(* IEC 61131-3 sources: std_i2980_v2.06_cp053/Source/IMM/ieccontrol/simulation (part 3) *)

(* ---- ABEasyMoldSimu.pu ---- *)
IMPORT_OVER_LISTFILE
 GET_REFTO
, EasyMold_Cmd
, tsCutOffCriterions

END_IMPORT

ALGORITHM_BLOCK ABEasyMoldSimu #DUMMY_EDIT_BLOCK

SYSTEM_VAR
 sv_MoldFullPosition : REAL;
 sv_MaxPressureSimu : REAL;
 sv_bAutoCycleRunning : BOOL;
 sv_ipCmd : REFTO EasyMold_Cmd;
 sv_CutOffParams : tsCutOffCriterions;
 sv_rScrewVolume : REAL;
 sv_rScrewDiameter : REAL;
 sv_rScrewPosition : REAL;
 sv_bEasyMoldTest : BOOL;
END_VAR

SYSTEM_OBJECT
 TaskSlow : TASK;
END_OBJECT

VAR
 uCounter : UDINT;
 rSAFactor : REAL;
 uTestCounter : UDINT := 0;
END_VAR

ALGORITHM EasyMoldWizardTest1

VAR_INPUT
 bRestart : BOOL := FALSE;
END_VAR

VAR_OUTPUT
 bReady : BOOL := FALSE;
END_VAR

VAR
 uCyclicCounter : UDINT := 0;
 uCyclicCounterPost : UDINT := 0;
 uCyclicLimit : UDINT := 2;
 uCyclicLimitTemp : UDINT := 2;
 rMaxPressSimu : REAL := 0.25;
 rMaxPressSimuPressLimit : REAL := 0.95;
 rDeltaPos : REAL := 0.0;
 rMoldFullPositionStart : REAL := 0.8;
 rMoldFullPositionStart1 : REAL := 0.2;
END_VAR
#BEGIN_EDIT_BLOCK
IF (rSAFactor <= 0.0) THEN
   rSAFactor := 1.0;
END_IF;
IF sv_rScrewVolume <= 0.0 THEN
   sv_MoldFullPosition :=  0.0;
   sv_MaxPressureSimu  :=  0.0;
   RETURN;
END_IF;
IF bRestart THEN
      bReady := FALSE;
      sv_MoldFullPosition := 0.001;//2.0 * sv_rScrewDiameter * 0.1 / sv_rScrewVolume;
      sv_MaxPressureSimu  := 0.05;
      uCyclicCounter      := 0;
      rDeltaPos           := 0.0;
ELSE
   IF sv_bAutoCycleRunning THEN

      CASE sv_ipCmd^ OF

         EMOLD_CMD_START: // Start
            bReady := FALSE;
            sv_MoldFullPosition := rMoldFullPositionStart;
            sv_MaxPressureSimu  :=  rMaxPressSimu;

         EMOLD_CMD_START1: // Start1
            sv_MoldFullPosition :=   rMoldFullPositionStart1;
            IF sv_MoldFullPosition >= ((sv_CutOffParams.rPositionThreshold / sv_rScrewVolume)- 0.1) THEN
                sv_MoldFullPosition := (sv_CutOffParams.rPositionThreshold - 0.11 * sv_rScrewVolume) / sv_rScrewVolume;
            END_IF;
            sv_MaxPressureSimu  :=  rMaxPressSimu;

         EMOLD_CMD_OPTIMIZE: // Optimize
            sv_MoldFullPosition :=  (sv_CutOffParams.rPositionThreshold - 0.01 * sv_rScrewVolume) / sv_rScrewVolume;
            IF sv_MoldFullPosition > rMoldFullPositionStart1 THEN
                rDeltaPos := sv_MoldFullPosition - rMoldFullPositionStart1;
                sv_MoldFullPosition := rMoldFullPositionStart1;
            END_IF;
            sv_MaxPressureSimu  :=  rMaxPressSimu;
            uCyclicCounter      :=  0;
            uCyclicCounterPost  := 0;

         EMOLD_CMD_CYCL_INJ:
//            IF uCyclicCounter = 0 THEN // 4
//               sv_MoldFullPosition := (0.95 * sv_rScrewVolume) / sv_rScrewVolume;
//               sv_MaxPressureSimu  := rMaxPressSimu;
//            ELSIF uCyclicCounter < uCyclicLimit THEN // 4
//               sv_MoldFullPosition := (sv_CutOffParams.rPositionThreshold + 0.01 * sv_rScrewVolume)  / sv_rScrewVolume;
//               sv_MaxPressureSimu  := rMaxPressSimu;
            IF uCyclicCounter = 0 THEN
               sv_MoldFullPosition := (sv_CutOffParams.rPositionThreshold - 0.01 * sv_rScrewVolume)  / sv_rScrewVolume - rDeltaPos;
               sv_MaxPressureSimu  := rMaxPressSimu;
            ELSIF uCyclicCounter < uCyclicLimit THEN
               sv_MoldFullPosition := (sv_CutOffParams.rPositionThreshold + 0.01 * sv_rScrewVolume)  / sv_rScrewVolume;
               sv_MaxPressureSimu  := rMaxPressSimuPressLimit;
            ELSIF uCyclicCounter < uCyclicLimit+uCyclicLimitTemp THEN
               sv_MoldFullPosition := (sv_CutOffParams.rPositionThreshold + 0.01 * sv_rScrewVolume)  / sv_rScrewVolume;
               sv_MaxPressureSimu  := rMaxPressSimu;
            ELSE
               sv_MoldFullPosition := (sv_CutOffParams.rPositionThreshold - 0.01 * sv_rScrewVolume)  / sv_rScrewVolume - rDeltaPos;
               sv_MaxPressureSimu  := rMaxPressSimu;
            END_IF;
            uCyclicCounter := uCyclicCounter +1;

         EMOLD_CMD_INC_MELTTEMP: //
            sv_MoldFullPosition := (sv_CutOffParams.rPositionThreshold - 0.01 * sv_rScrewVolume) / sv_rScrewVolume - rDeltaPos;
            sv_MaxPressureSimu  := rMaxPressSimu;

         EMOLD_CMD_INC_MOLDTEMP: // CyclicInject 1: 1. Durchlauf
            sv_MoldFullPosition := (sv_CutOffParams.rPositionThreshold - 0.01 * sv_rScrewVolume) / sv_rScrewVolume - rDeltaPos;
            sv_MaxPressureSimu  := rMaxPressSimu;

         EMOLD_CMD_POSTCUTOFF:
//            IF (uCyclicCounterPost=0) THEN
//               sv_MoldFullPosition := (0.95 * sv_rScrewVolume) / sv_rScrewVolume;
//               sv_MaxPressureSimu  := rMaxPressSimu;
//               uCyclicCounter      :=  0;
//                uCyclicCounterPost := 1;
//            ELSE
                sv_MoldFullPosition := (sv_CutOffParams.rPositionThreshold - 0.01 * sv_rScrewVolume) / sv_rScrewVolume - rDeltaPos;
                sv_MaxPressureSimu  := rMaxPressSimu;
                uCyclicCounter      := 0;
//            END_IF;

         EMOLD_CMD_INC_PACKPRESS:
            sv_MoldFullPosition := (sv_CutOffParams.rPositionThreshold - 0.01 * sv_rScrewVolume) / sv_rScrewVolume - rDeltaPos;
            sv_MaxPressureSimu  := rMaxPressSimuPressLimit;

         EMOLD_CMD_CORR_MELTCUS:
            sv_MoldFullPosition := (sv_CutOffParams.rPositionThreshold - 0.01 * sv_rScrewVolume) / sv_rScrewVolume - rDeltaPos;
            sv_MaxPressureSimu  := rMaxPressSimu;
            bReady := TRUE;

         EMOLD_CMD_HOTRUNNER: //
            sv_MoldFullPosition := (sv_CutOffParams.rPositionThreshold - 0.01 * sv_rScrewVolume) / sv_rScrewVolume - rDeltaPos;
            sv_MaxPressureSimu  := rMaxPressSimu;

      ELSE
            // default state
            bReady := FALSE;
            sv_MoldFullPosition := (sv_CutOffParams.rPositionThreshold - 0.01 * sv_rScrewVolume) / sv_rScrewVolume - rDeltaPos;
            sv_MaxPressureSimu  := rMaxPressSimu;

      END_CASE;
      uCounter := uCounter+1;
   ELSE
      sv_MoldFullPosition := sv_rScrewDiameter * 0.1 / sv_rScrewVolume;
      sv_MaxPressureSimu  := 50.0;
   END_IF;
   IF (sv_MoldFullPosition < 0.001) THEN
       sv_MoldFullPosition := 0.001;
   END_IF;
END_IF;
IF sv_MoldFullPosition > 1.0 THEN
   sv_MoldFullPosition := 1.0;
END_IF;

;#END_EDIT_BLOCK END_ALGORITHM

POSTUPDATE_ALGORITHM puEasyMoldWizardTestStart ON TaskSlow WITH sv_bEasyMoldTest

#BEGIN_EDIT_BLOCK

IF sv_bEasyMoldTest THEN
   uCounter := 1;
   rSAFactor := sv_rScrewDiameter * sv_rScrewDiameter * cEMW_Pi * 0.25e-3;
   sv_rScrewPosition := sv_rScrewDiameter * rSAFactor;
   uTestCounter := 0;
   START_PROCESS_ALGORITHM(paRunAlgo);
END_IF;

;#END_EDIT_BLOCK END_ALGORITHM

POSTUPDATE_ALGORITHM puEasyMoldWizardTestRun ON TaskSlow WITH sv_bAutoCycleRunning

#BEGIN_EDIT_BLOCK
IF sv_bEasyMoldTest THEN
    //piCmd := @sv_iCmd;
    START_PROCESS_ALGORITHM(paRunAlgo);
END_IF;

;#END_EDIT_BLOCK END_ALGORITHM

PROCESS_ALGORITHM paRunAlgo ON TaskSlow

#BEGIN_EDIT_BLOCK
CASE uTestCounter OF
   0:
      EasyMoldWizardTest1(bRestart:=TRUE);
      uTestCounter := uTestCounter + 1;

   1: // EasyMoldWizardTest1
      EasyMoldWizardTest1(bRestart:=FALSE);

ELSE
   // EasyMoldWizardTest1
   EasyMoldWizardTest1();
   uTestCounter := 1;
END_CASE;

STOP_PROCESS_ALGORITHM();

;#END_EDIT_BLOCK END_ALGORITHM

END_ALGORITHM_BLOCK

#END_OF_IEC_PART

@Puma @IecEditor 6 97 @Pou 25
@@@BEG_Comment@@@

@@@END_Comment@@@

@BEG_Contents

@BEG_Func
@RT(17)FuncTreeContainer
1
@Var @RT(9)GET_REFTO @RT(0) @T @T @DERIVED 0 @F @RT(22)KEBA_STANDARD_FUNCTION @F
@T
@BEG_Attrib
0 @RT(0) @RT(0)
@END_Attrib
1 1 @F @F @F @F

@END_Func

@BEG_Const
@RT(18)ConstTreeContainer
0
@END_Const

@BEG_Export

@BEG_Kind
@ALGORITHM_BLOCK @RT(14)ABEasyMoldSimu @STRUCTURED_TEXT
@RT(0) @RT(0) @RT(0)
@END_Kind

@BEG_Dcl
@RT(16)DclTreeContainer
13
@Var @RT(8)TaskSlow @RT(0) @T @F @DT @RT(4)TASK @RT(0) @T @T @BASIC 0 @F
@F @F
@T
@BEG_Attrib
3 @RT(0) @RT(0) @RT(0)
@END_Attrib
1 7 @F @F @F @F

@Var @RT(19)sv_MoldFullPosition @RT(0) @T @F @DT @RT(4)REAL @RT(0) @T @T @BASIC 0 @F
@F @F
@T
@BEG_Attrib
3 @RT(0) @RT(0) @RT(0)
@END_Attrib
1 8 @F @F @F @F

@Var @RT(18)sv_MaxPressureSimu @RT(0) @T @F @DT @RT(4)REAL @RT(0) @T @T @BASIC 0 @F
@F @F
@T
@BEG_Attrib
3 @RT(0) @RT(0) @RT(0)
@END_Attrib
1 8 @F @F @F @F

@Var @RT(20)sv_bAutoCycleRunning @RT(0) @T @F @DT @RT(4)BOOL @RT(0) @T @T @BASIC 0 @F
@F @F
@T
@BEG_Attrib
3 @RT(0) @RT(0) @RT(0)
@END_Attrib
1 8 @F @F @F @F

@Var @RT(8)sv_ipCmd @RT(0) @T @T @REFTO 0 @F @DERIVED 0 @T @T @DT @RT(12)EasyMold_Cmd @RT(0) @T @T @UNKNOWN 0 @F
@F @F
@T
@BEG_Attrib
3 @RT(0) @RT(0) @RT(0)
@END_Attrib
1 8 @F @F @F @F

@Var @RT(15)sv_CutOffParams @RT(0) @T @T @DERIVED 0 @T @T @DT @RT(18)tsCutOffCriterions @RT(0) @T @T @UNKNOWN 0 @F
@F @F
@T
@BEG_Attrib
3 @RT(0) @RT(0) @RT(0)
@END_Attrib
1 8 @F @F @F @F

@Var @RT(15)sv_rScrewVolume @RT(0) @T @F @DT @RT(4)REAL @RT(0) @T @T @BASIC 0 @F
@F @F
@T
@BEG_Attrib
3 @RT(0) @RT(0) @RT(0)
@END_Attrib
1 8 @F @F @F @F

@Var @RT(8)uCounter @RT(0) @T @F @DT @RT(5)UDINT @RT(0) @T @T @BASIC 0 @F
@F @F
@T
@BEG_Attrib
3 @RT(0) @RT(0) @RT(0)
@END_Attrib
1 0 @F @F @F @F

@Var @RT(17)sv_rScrewDiameter @RT(0) @T @F @DT @RT(4)REAL @RT(0) @T @T @BASIC 0 @F
@F @F
@T
@BEG_Attrib
3 @RT(0) @RT(0) @RT(0)
@END_Attrib
1 8 @F @F @F @F

@Var @RT(9)rSAFactor @RT(0) @T @F @DT @RT(4)REAL @RT(0) @T @T @BASIC 0 @F
@F @F
@T
@BEG_Attrib
3 @RT(0) @RT(0) @RT(0)
@END_Attrib
1 0 @F @F @F @F

@Var @RT(17)sv_rScrewPosition @RT(0) @T @F @DT @RT(4)REAL @RT(0) @T @T @BASIC 0 @F
@F @F
@T
@BEG_Attrib
3 @RT(0) @RT(0) @RT(0)
@END_Attrib
1 8 @F @F @F @F

@Var @RT(16)sv_bEasyMoldTest @RT(0) @T @F @DT @RT(4)BOOL @RT(0) @T @T @BASIC 0 @F
@F @F
@T
@BEG_Attrib
3 @RT(0) @RT(0) @RT(0)
@END_Attrib
1 8 @F @F @F @F

@Var @RT(12)uTestCounter @RT(0) @T @F @DT @RT(5)UDINT @RT(0) @T @T @BASIC 0 @F
@F @F
@T
@BEG_Attrib
3 @RT(1)0 @RT(0) @RT(0)
@END_Attrib
1 0 @F @F @F @F

@END_Dcl

@END_Export

@BEG_Body

4

@BEG_Export

@BEG_Algo
@ALGORITHM @RT(19)EasyMoldWizardTest1 @STRUCTURED_TEXT
@RT(0) @RT(0) @RT(0) @F @F
@END_Algo

@BEG_Dcl
@RT(16)DclTreeContainer
11
@Var @RT(8)bRestart @RT(0) @T @F @DT @RT(4)BOOL @RT(0) @T @T @BASIC 0 @F
@F @F
@T
@BEG_Attrib
3 @RT(5)FALSE @RT(0) @RT(0)
@END_Attrib
1 1 @F @F @F @F

@Var @RT(6)bReady @RT(0) @T @F @DT @RT(4)BOOL @RT(0) @T @T @BASIC 0 @F
@F @F
@T
@BEG_Attrib
3 @RT(5)FALSE @RT(0) @RT(0)
@END_Attrib
1 3 @F @F @F @F

@Var @RT(14)uCyclicCounter @RT(0) @T @F @DT @RT(5)UDINT @RT(0) @T @T @BASIC 0 @F
@F @F
@T
@BEG_Attrib
3 @RT(1)0 @RT(0) @RT(0)
@END_Attrib
1 0 @F @F @F @F

@Var @RT(18)uCyclicCounterPost @RT(0) @T @F @DT @RT(5)UDINT @RT(0) @T @T @BASIC 0 @F
@F @F
@T
@BEG_Attrib
3 @RT(1)0 @RT(0) @RT(0)
@END_Attrib
1 0 @F @F @F @F

@Var @RT(12)uCyclicLimit @RT(0) @T @F @DT @RT(5)UDINT @RT(0) @T @T @BASIC 0 @F
@F @F
@T
@BEG_Attrib
3 @RT(1)2 @RT(0) @RT(0)
@END_Attrib
1 0 @F @F @F @F

@Var @RT(16)uCyclicLimitTemp @RT(0) @T @F @DT @RT(5)UDINT @RT(0) @T @T @BASIC 0 @F
@F @F
@T
@BEG_Attrib
3 @RT(1)2 @RT(0) @RT(0)
@END_Attrib
1 0 @F @F @F @F

@Var @RT(13)rMaxPressSimu @RT(0) @T @F @DT @RT(4)REAL @RT(0) @T @T @BASIC 0 @F
@F @F
@T
@BEG_Attrib
3 @RT(4)0.25 @RT(0) @RT(0)
@END_Attrib
1 0 @F @F @F @F

@Var @RT(23)rMaxPressSimuPressLimit @RT(0) @T @F @DT @RT(4)REAL @RT(0) @T @T @BASIC 0 @F
@F @F
@T
@BEG_Attrib
3 @RT(4)0.95 @RT(0) @RT(0)
@END_Attrib
1 0 @F @F @F @F

@Var @RT(9)rDeltaPos @RT(0) @T @F @DT @RT(4)REAL @RT(0) @T @T @BASIC 0 @F
@F @F
@T
@BEG_Attrib
3 @RT(3)0.0 @RT(0) @RT(0)
@END_Attrib
1 0 @F @F @F @F

@Var @RT(22)rMoldFullPositionStart @RT(0) @T @F @DT @RT(4)REAL @RT(0) @T @T @BASIC 0 @F
@F @F
@T
@BEG_Attrib
3 @RT(3)0.8 @RT(0) @RT(0)
@END_Attrib
1 0 @F @F @F @F

@Var @RT(23)rMoldFullPositionStart1 @RT(0) @T @F @DT @RT(4)REAL @RT(0) @T @T @BASIC 0 @F
@F @F
@T
@BEG_Attrib
3 @RT(3)0.2 @RT(0) @RT(0)
@END_Attrib
1 0 @F @F @F @F

@END_Dcl

@END_Export

@BEG_Export

@BEG_Algo
@POSTUPDATE_ALGORITHM @RT(25)puEasyMoldWizardTestStart @STRUCTURED_TEXT
@RT(0) @RT(16)sv_bEasyMoldTest @RT(8)TaskSlow @F @F
@END_Algo

@BEG_Dcl
@RT(16)DclTreeContainer
0
@END_Dcl

@END_Export

@BEG_Export

@BEG_Algo
@POSTUPDATE_ALGORITHM @RT(23)puEasyMoldWizardTestRun @STRUCTURED_TEXT
@RT(0) @RT(20)sv_bAutoCycleRunning @RT(8)TaskSlow @F @F
@END_Algo

@BEG_Dcl
@RT(16)DclTreeContainer
0
@END_Dcl

@END_Export

@BEG_Export

@BEG_Algo
@PROCESS_ALGORITHM @RT(9)paRunAlgo @STRUCTURED_TEXT
@RT(0) @RT(0) @RT(8)TaskSlow @F @F
@END_Algo

@BEG_Dcl
@RT(16)DclTreeContainer
0
@END_Dcl

@END_Export

@BEG_Body
@TL(117)
IF (rSAFactor <= 0.0) THEN
   rSAFactor := 1.0;
END_IF;
IF sv_rScrewVolume <= 0.0 THEN
   sv_MoldFullPosition :=  0.0;
   sv_MaxPressureSimu  :=  0.0;
   RETURN;
END_IF;
IF bRestart THEN
      bReady := FALSE;
      sv_MoldFullPosition := 0.001;//2.0 * sv_rScrewDiameter * 0.1 / sv_rScrewVolume;
      sv_MaxPressureSimu  := 0.05;
      uCyclicCounter      := 0;
      rDeltaPos           := 0.0;
ELSE
   IF sv_bAutoCycleRunning THEN

      CASE sv_ipCmd^ OF

         EMOLD_CMD_START: // Start
            bReady := FALSE;
            sv_MoldFullPosition := rMoldFullPositionStart;
            sv_MaxPressureSimu  :=  rMaxPressSimu;

         EMOLD_CMD_START1: // Start1
            sv_MoldFullPosition :=   rMoldFullPositionStart1;
            IF sv_MoldFullPosition >= ((sv_CutOffParams.rPositionThreshold / sv_rScrewVolume)- 0.1) THEN
                sv_MoldFullPosition := (sv_CutOffParams.rPositionThreshold - 0.11 * sv_rScrewVolume) / sv_rScrewVolume;
            END_IF;
            sv_MaxPressureSimu  :=  rMaxPressSimu;

         EMOLD_CMD_OPTIMIZE: // Optimize
            sv_MoldFullPosition :=  (sv_CutOffParams.rPositionThreshold - 0.01 * sv_rScrewVolume) / sv_rScrewVolume;
            IF sv_MoldFullPosition > rMoldFullPositionStart1 THEN
                rDeltaPos := sv_MoldFullPosition - rMoldFullPositionStart1;
                sv_MoldFullPosition := rMoldFullPositionStart1;
            END_IF;
            sv_MaxPressureSimu  :=  rMaxPressSimu;
            uCyclicCounter      :=  0;
            uCyclicCounterPost  := 0;

         EMOLD_CMD_CYCL_INJ:
//            IF uCyclicCounter = 0 THEN // 4
//               sv_MoldFullPosition := (0.95 * sv_rScrewVolume) / sv_rScrewVolume;
//               sv_MaxPressureSimu  := rMaxPressSimu;
//            ELSIF uCyclicCounter < uCyclicLimit THEN // 4
//               sv_MoldFullPosition := (sv_CutOffParams.rPositionThreshold + 0.01 * sv_rScrewVolume)  / sv_rScrewVolume;
//               sv_MaxPressureSimu  := rMaxPressSimu;
            IF uCyclicCounter = 0 THEN
               sv_MoldFullPosition := (sv_CutOffParams.rPositionThreshold - 0.01 * sv_rScrewVolume)  / sv_rScrewVolume - rDeltaPos;
               sv_MaxPressureSimu  := rMaxPressSimu;
            ELSIF uCyclicCounter < uCyclicLimit THEN
               sv_MoldFullPosition := (sv_CutOffParams.rPositionThreshold + 0.01 * sv_rScrewVolume)  / sv_rScrewVolume;
               sv_MaxPressureSimu  := rMaxPressSimuPressLimit;
            ELSIF uCyclicCounter < uCyclicLimit+uCyclicLimitTemp THEN
               sv_MoldFullPosition := (sv_CutOffParams.rPositionThreshold + 0.01 * sv_rScrewVolume)  / sv_rScrewVolume;
               sv_MaxPressureSimu  := rMaxPressSimu;
            ELSE
               sv_MoldFullPosition := (sv_CutOffParams.rPositionThreshold - 0.01 * sv_rScrewVolume)  / sv_rScrewVolume - rDeltaPos;
               sv_MaxPressureSimu  := rMaxPressSimu;
            END_IF;
            uCyclicCounter := uCyclicCounter +1;

         EMOLD_CMD_INC_MELTTEMP: //
            sv_MoldFullPosition := (sv_CutOffParams.rPositionThreshold - 0.01 * sv_rScrewVolume) / sv_rScrewVolume - rDeltaPos;
            sv_MaxPressureSimu  := rMaxPressSimu;

         EMOLD_CMD_INC_MOLDTEMP: // CyclicInject 1: 1. Durchlauf
            sv_MoldFullPosition := (sv_CutOffParams.rPositionThreshold - 0.01 * sv_rScrewVolume) / sv_rScrewVolume - rDeltaPos;
            sv_MaxPressureSimu  := rMaxPressSimu;

         EMOLD_CMD_POSTCUTOFF:
//            IF (uCyclicCounterPost=0) THEN
//               sv_MoldFullPosition := (0.95 * sv_rScrewVolume) / sv_rScrewVolume;
//               sv_MaxPressureSimu  := rMaxPressSimu;
//               uCyclicCounter      :=  0;
//                uCyclicCounterPost := 1;
//            ELSE
                sv_MoldFullPosition := (sv_CutOffParams.rPositionThreshold - 0.01 * sv_rScrewVolume) / sv_rScrewVolume - rDeltaPos;
                sv_MaxPressureSimu  := rMaxPressSimu;
                uCyclicCounter      := 0;
//            END_IF;

         EMOLD_CMD_INC_PACKPRESS:
            sv_MoldFullPosition := (sv_CutOffParams.rPositionThreshold - 0.01 * sv_rScrewVolume) / sv_rScrewVolume - rDeltaPos;
            sv_MaxPressureSimu  := rMaxPressSimuPressLimit;

         EMOLD_CMD_CORR_MELTCUS:
            sv_MoldFullPosition := (sv_CutOffParams.rPositionThreshold - 0.01 * sv_rScrewVolume) / sv_rScrewVolume - rDeltaPos;
            sv_MaxPressureSimu  := rMaxPressSimu;
            bReady := TRUE;

         EMOLD_CMD_HOTRUNNER: //
            sv_MoldFullPosition := (sv_CutOffParams.rPositionThreshold - 0.01 * sv_rScrewVolume) / sv_rScrewVolume - rDeltaPos;
            sv_MaxPressureSimu  := rMaxPressSimu;

      ELSE
            // default state
            bReady := FALSE;
            sv_MoldFullPosition := (sv_CutOffParams.rPositionThreshold - 0.01 * sv_rScrewVolume) / sv_rScrewVolume - rDeltaPos;
            sv_MaxPressureSimu  := rMaxPressSimu;

      END_CASE;
      uCounter := uCounter+1;
   ELSE
      sv_MoldFullPosition := sv_rScrewDiameter * 0.1 / sv_rScrewVolume;
      sv_MaxPressureSimu  := 50.0;
   END_IF;
   IF (sv_MoldFullPosition < 0.001) THEN
       sv_MoldFullPosition := 0.001;
   END_IF;
END_IF;
IF sv_MoldFullPosition > 1.0 THEN
   sv_MoldFullPosition := 1.0;
END_IF;

@END_Body

@@@BEG_Comment@@@
@TL(0)

@@@END_Comment@@@

@BEG_Body
@TL(9)

IF sv_bEasyMoldTest THEN
   uCounter := 1;
   rSAFactor := sv_rScrewDiameter * sv_rScrewDiameter * cEMW_Pi * 0.25e-3;
   sv_rScrewPosition := sv_rScrewDiameter * rSAFactor;
   uTestCounter := 0;
   START_PROCESS_ALGORITHM(paRunAlgo);
END_IF;

@END_Body

@@@BEG_Comment@@@
@TL(0)

@@@END_Comment@@@

@BEG_Body
@TL(5)
IF sv_bEasyMoldTest THEN
    //piCmd := @sv_iCmd;
    START_PROCESS_ALGORITHM(paRunAlgo);
END_IF;

@END_Body

@@@BEG_Comment@@@
@TL(0)

@@@END_Comment@@@

@BEG_Body
@TL(16)
CASE uTestCounter OF
   0:
      EasyMoldWizardTest1(bRestart:=TRUE);
      uTestCounter := uTestCounter + 1;

   1: // EasyMoldWizardTest1
      EasyMoldWizardTest1(bRestart:=FALSE);

ELSE
   // EasyMoldWizardTest1
   EasyMoldWizardTest1();
   uTestCounter := 1;
END_CASE;

STOP_PROCESS_ALGORITHM();

@END_Body

@@@BEG_Comment@@@
@TL(0)

@@@END_Comment@@@
@END_Body

@END_Contents

(* ---- ABEjeSimu.pu ---- *)
IMPORT_OVER_LISTFILE
 GET_TASK_INTERVAL
, GET_SYNC_REFTO
, KSYS_Status_OK
, FBEPForceAI
, FBEPForceDI
, FBEPUnForceAI
, FBEPUnForceDI
, tsRequiredPumps
, FBGetSimulationSource
, TON
, KSYS_Status
, FBGetRequiredPumps

END_IMPORT

ALGORITHM_BLOCK ABEjeSimu #DUMMY_EDIT_BLOCK

SYSTEM_VAR
 sv_bSimulate : BOOL;
 sv_bInitStart : BOOL;
 ai_Position_stat : BOOL;
 sv_ForceEjectorBack : BOOL;
 sv_bInitDone : BOOL;
END_VAR

SYSTEM_OBJECT
 TaskSim : TASK;
 PU_Task_13 : TASK;
 TaskAnalog : TASK;
END_OBJECT

VAR
 fbEPForceAI : FBEPForceAI;
 fbEPForceDI : FBEPForceDI;
 mbDIEjectorBackLinked : BOOL;
 fbEPUnForceAI : FBEPUnForceAI;
 fbEPUnForceDI : FBEPUnForceDI;
 mpPumps : REFTO tsRequiredPumps;
 mprVelocity : REFTO REAL;
 fbGetSimulationSource : FBGetSimulationSource;
END_VAR

POSTUPDATE_ALGORITHM pStart ON PU_Task_13 WITH sv_bSimulate,sv_bInitStart

#BEGIN_EDIT_BLOCK
(**************************************** WARNING ********************************************
 *** The KEBA Kemro K2 System including software is not intended for safety control tasks! ***
 ***                       For further information see Comment tab!                        ***
 *********************************************************************************************)

IF sv_bSimulate THEN
   START_PROCESS_ALGORITHM(paSimulate);
END_IF;

;#END_EDIT_BLOCK END_ALGORITHM

PROCESS_ALGORITHM paSimulate ON TaskAnalog

VAR
 rEjectDivision : REAL := 0.3;
 mrEjectorPosRaw : REAL;
 rEjectTimeFor10V : REAL := 1.0;
 TimerFwd : TON (* chad(CR_0038565) *);
 TimerBwd : TON (* chad(CR_0038565) *);
 rCycleTime : REAL;
 dCycleTime : TIME;
 prEjectorPosRaw : REFTO REAL;
 bAIEjectorTransLinked : BOOL;
 pbDOEjectorBwd : REFTO BOOL;
 pbDOEjectorFwd : REFTO BOOL;
 bDOEjectorFwdLinked : BOOL;
 bDOEjectorBwdLinked : BOOL;
 bDIEjectorFwdLinked : BOOL (* chad(CR_0038565) *);
 pbDummy : REFTO BOOL;
 Status : KSYS_Status;
 bDIEjectorSafetyPlateLinked : BOOL;
END_VAR

(* IecGraph-Code *)

(* init step *)
INITIAL_STEP INIT:
aInit (P);
END_STEP

(* steps *)
STEP SIM:
aSimulate (N);
END_STEP

STEP STOP:
aStopSimu (P);
END_STEP

(* transitions *)
TRANSITION SimRequired (* SimRequired *) FROM INIT TO SIM :=  #BEGIN_EDIT_BLOCK
sv_bSimulate
;#END_EDIT_BLOCK
END_TRANSITION

TRANSITION StpSimRequired (* StpSimRequired *) FROM SIM TO STOP :=  #BEGIN_EDIT_BLOCK
NOT sv_bSimulate
;#END_EDIT_BLOCK
END_TRANSITION

TRANSITION Return (* Return *) FROM STOP TO SIM :=  #BEGIN_EDIT_BLOCK
TRUE
;#END_EDIT_BLOCK
END_TRANSITION

(* end IecGraph-Code *)
(* sfc-code *)

(* stand alone actions *)
ACTION aInit: #BEGIN_EDIT_BLOCK
(**************************************** WARNING ********************************************
 *** The KEBA Kemro K2 System including software is not intended for safety control tasks! ***
 ***                       For further information see Comment tab!                        ***
 *********************************************************************************************)

pbDummy := GET_SYNC_REFTO('Ejector1.di_EjectorBwd', T#0s, Status);
mbDIEjectorBackLinked := (Status = KSYS_Status_OK);

pbDummy := GET_SYNC_REFTO('Ejector1.di_EjectorFwd', T#0s, Status);
bDIEjectorFwdLinked := (Status = KSYS_Status_OK);

prEjectorPosRaw := GET_SYNC_REFTO('Ejector1.ai_Position', T#0s, Status);
bAIEjectorTransLinked := (Status = KSYS_Status_OK);

pbDOEjectorFwd := GET_SYNC_REFTO('Ejector1.do_Forward', T#0s, Status);
bDOEjectorFwdLinked := (Status = KSYS_Status_OK);

pbDOEjectorBwd := GET_SYNC_REFTO('Ejector1.do_Backward', T#0s, Status);
bDOEjectorBwdLinked := (Status = KSYS_Status_OK);

pbDummy := GET_SYNC_REFTO('Ejector1.di_SafetyPlate', T#0s, Status);
bDIEjectorSafetyPlateLinked := (Status = KSYS_Status_OK);
IF bDIEjectorSafetyPlateLinked THEN
   fbEPForceDI(sSysVar := 'Ejector1.di_SafetyPlate',Value := TRUE);
END_IF;

dCycleTime :=  GET_TASK_INTERVAL();
rCycleTime := (LINT_TO_REAL(TIME_TO_LINT(dCycleTime))) / 1000000.0;
rEjectDivision := 1.0  / rEjectTimeFor10V * rCycleTime;

sv_ForceEjectorBack := TRUE;

IF bDIEjectorFwdLinked THEN    //chad(CR_0038565)
   fbEPForceDI(sSysVar := 'Ejector1.di_EjectorFwd',Value := FALSE);
END_IF;

IF bAIEjectorTransLinked THEN
   ai_Position_stat := FALSE;
   fbEPForceAI(sSysVar := 'Ejector1.ai_Position',Value := 0.0, Range := 10.0);
END_IF;

;#END_EDIT_BLOCK END_ACTION (*aInit*)
ACTION aSimulate: #BEGIN_EDIT_BLOCK
(**************************************** WARNING ********************************************
 *** The KEBA Kemro K2 System including software is not intended for safety control tasks! ***
 ***                       For further information see Comment tab!                        ***
 *********************************************************************************************)

IF bAIEjectorTransLinked THEN
   IF bDOEjectorFwdLinked AND pbDOEjectorFwd^ THEN
      mrEjectorPosRaw := prEjectorPosRaw^ + MUL(rEjectDivision,mprVelocity^);
      sv_ForceEjectorBack := FALSE;
   ELSIF bDOEjectorBwdLinked AND pbDOEjectorBwd^ THEN
      mrEjectorPosRaw := prEjectorPosRaw^ - MUL(rEjectDivision,mprVelocity^);
      IF prEjectorPosRaw^ <= 2.0 THEN
            sv_ForceEjectorBack := TRUE;
      END_IF;
   END_IF;
   fbEPForceAI(sSysVar := 'Ejector1.ai_Position', Value := MAX(mrEjectorPosRaw,0.0), Range := 10.0);

ELSE    //chad(CR_0038565) - transducer not linked

   //Move forward simulation
   IF bDOEjectorFwdLinked AND (NOT pbDOEjectorFwd^) THEN
      TimerFwd(IN := FALSE);
   END_IF;

   IF bDOEjectorFwdLinked AND pbDOEjectorFwd^ THEN
      TimerFwd(IN := TRUE, PT := t#4s);
      IF mbDIEjectorBackLinked THEN
         sv_ForceEjectorBack := FALSE;
         TimerBwd(IN := FALSE);
      END_IF;

      IF TimerFwd.Q AND bDIEjectorFwdLinked THEN
         fbEPForceDI(sSysVar := 'Ejector1.di_EjectorFwd',Value := TRUE);
         TimerFwd(IN := FALSE);
      END_IF;
   END_IF;

   //Move backward simulation
   IF bDOEjectorBwdLinked AND (NOT pbDOEjectorBwd^) THEN
      TimerBwd(IN := FALSE);
   END_IF;

   IF bDOEjectorBwdLinked AND pbDOEjectorBwd^ THEN
      TimerBwd(IN := TRUE, PT := t#4s);
      IF bDIEjectorFwdLinked THEN
         fbEPForceDI(sSysVar := 'Ejector1.di_EjectorFwd',Value := FALSE);
         TimerFwd(IN := FALSE);
      END_IF;

      IF TimerBwd.Q AND mbDIEjectorBackLinked THEN
         sv_ForceEjectorBack := TRUE;
         TimerBwd(IN := FALSE);
      END_IF;
   END_IF;
END_IF;

;#END_EDIT_BLOCK END_ACTION (*aSimulate*)
ACTION aStopSimu: #BEGIN_EDIT_BLOCK
(**************************************** WARNING ********************************************
 *** The KEBA Kemro K2 System including software is not intended for safety control tasks! ***
 ***                       For further information see Comment tab!                        ***
 *********************************************************************************************)

IF bAIEjectorTransLinked THEN
   fbEPUnForceAI(sSysVar := 'Ejector1.ai_Position');
END_IF;
IF mbDIEjectorBackLinked THEN
   fbEPUnForceDI(sSysVar := 'Ejector1.di_EjectorBwd');
END_IF;
IF bDIEjectorSafetyPlateLinked THEN
   fbEPUnForceDI(sSysVar := 'Ejector1.di_SafetyPlate');
END_IF;
IF bDIEjectorFwdLinked THEN   //chad(CR_0038565)
   fbEPUnForceDI(sSysVar := 'Ejector1.di_EjectorFwd');
END_IF;

STOP_PROCESS_ALGORITHM();

;#END_EDIT_BLOCK END_ACTION (*aStopSimu*)
(* end sfc-code *)

END_ALGORITHM

POSTUPDATE_ALGORITHM pEjectorBwd ON TaskSim WITH sv_ForceEjectorBack

#BEGIN_EDIT_BLOCK
(**************************************** WARNING ********************************************
 *** The KEBA Kemro K2 System including software is not intended for safety control tasks! ***
 ***                       For further information see Comment tab!                        ***
 *********************************************************************************************)

IF mbDIEjectorBackLinked THEN
   fbEPForceDI(sSysVar := 'Ejector1.di_EjectorBwd',Value := sv_ForceEjectorBack);
END_IF;

;#END_EDIT_BLOCK END_ALGORITHM

ALGORITHM aGetSimulationSource

#BEGIN_EDIT_BLOCK
(**************************************** WARNING ********************************************
 *** The KEBA Kemro K2 System including software is not intended for safety control tasks! ***
 ***                       For further information see Comment tab!                        ***
 *********************************************************************************************)

fbGetSimulationSource(pRequiredPumps := mpPumps,
                      prVelocity => mprVelocity);

;#END_EDIT_BLOCK END_ALGORITHM

POSTUPDATE_ALGORITHM pInitDone ON TaskSim WITH sv_bInitDone

VAR
 fbGetRequiredPumps : FBGetRequiredPumps;
END_VAR
#BEGIN_EDIT_BLOCK
(**************************************** WARNING ********************************************
 *** The KEBA Kemro K2 System including software is not intended for safety control tasks! ***
 ***                       For further information see Comment tab!                        ***
 *********************************************************************************************)

//get required pumps
fbGetRequiredPumps.DeviceId.CompId := cCompEjector;
fbGetRequiredPumps.DeviceId.IndexId := 1;

fbGetRequiredPumps(MoveDir := cMoveFwd,
                   MoveId := cMoveFwd);
mpPumps := fbGetRequiredPumps.pPumps;

aGetSimulationSource();

;#END_EDIT_BLOCK END_ALGORITHM

POSTUPDATE_ALGORITHM pRequiredPumps ON TaskSim WITH mpPumps^.RequiredPumps

#BEGIN_EDIT_BLOCK
(**************************************** WARNING ********************************************
 *** The KEBA Kemro K2 System including software is not intended for safety control tasks! ***
 ***                       For further information see Comment tab!                        ***
 *********************************************************************************************)

aGetSimulationSource();

;#END_EDIT_BLOCK END_ALGORITHM

END_ALGORITHM_BLOCK

#END_OF_IEC_PART

@Puma @IecEditor 6 113 @Pou 25
@@@BEG_Comment@@@

@@@END_Comment@@@

@BEG_Contents

@BEG_Func
@RT(17)FuncTreeContainer
2
@Var @RT(17)GET_TASK_INTERVAL @RT(0) @T @T @DERIVED 0 @F @RT(22)KEBA_STANDARD_FUNCTION @F
@T
@BEG_Attrib
0 @RT(0) @RT(0)
@END_Attrib
1 1 @F @F @F @F

@Var @RT(14)GET_SYNC_REFTO @RT(0) @T @T @DERIVED 0 @F @RT(22)KEBA_STANDARD_FUNCTION @F
@T
@BEG_Attrib
0 @RT(0) @RT(0)
@END_Attrib
1 1 @F @F @F @F

@END_Func

@BEG_Const
@RT(18)ConstTreeContainer
1
@Var @RT(14)KSYS_Status_OK @RT(0) @T @T @DERIVED 0 @F @RT(11)KSYS_Status @F
@T
@BEG_Attrib
0 @RT(1)1 @RT(0)
@END_Attrib
1 1 @F @F @F @F

@END_Const

@BEG_Export

@BEG_Kind
@ALGORITHM_BLOCK @RT(9)ABEjeSimu @STRUCTURED_TEXT
@RT(0) @RT(0) @RT(0)
@END_Kind

@BEG_Dcl
@RT(16)DclTreeContainer
16
@Var @RT(12)sv_bSimulate @RT(0) @T @F @DT @RT(4)BOOL @RT(0) @T @T @BASIC 0 @F
@F @F
@T
@BEG_Attrib
3 @RT(0) @RT(0) @RT(0)
@END_Attrib
1 8 @F @F @F @F

@Var @RT(13)sv_bInitStart @RT(0) @T @F @DT @RT(4)BOOL @RT(0) @T @T @BASIC 0 @F
@F @F
@T
@BEG_Attrib
3 @RT(0) @RT(0) @RT(0)
@END_Attrib
1 8 @F @F @F @F

@Var @RT(16)ai_Position_stat @RT(0) @T @F @DT @RT(4)BOOL @RT(0) @T @T @BASIC 0 @F
@F @F
@T
@BEG_Attrib
3 @RT(0) @RT(0) @RT(0)
@END_Attrib
1 8 @F @F @F @F

@Var @RT(7)TaskSim @RT(0) @T @F @DT @RT(4)TASK @RT(0) @T @T @BASIC 0 @F
@F @F
@T
@BEG_Attrib
3 @RT(0) @RT(0) @RT(0)
@END_Attrib
1 7 @F @F @F @F

@Var @RT(10)PU_Task_13 @RT(0) @T @F @DT @RT(4)TASK @RT(0) @T @T @BASIC 0 @F
@F @F
@T
@BEG_Attrib
3 @RT(0) @RT(0) @RT(0)
@END_Attrib
1 7 @F @F @F @F

@Var @RT(11)fbEPForceAI @RT(0) @T @T @DERIVED 0 @T @T @DT @RT(11)FBEPForceAI @RT(0) @T @T @UNKNOWN 0 @F
@F @F
@T
@BEG_Attrib
3 @RT(0) @RT(0) @RT(0)
@END_Attrib
1 0 @F @F @F @F

@Var @RT(11)fbEPForceDI @RT(0) @T @T @DERIVED 0 @T @T @DT @RT(11)FBEPForceDI @RT(0) @T @T @UNKNOWN 0 @F
@F @F
@T
@BEG_Attrib
3 @RT(0) @RT(0) @RT(0)
@END_Attrib
1 0 @F @F @F @F

@Var @RT(21)mbDIEjectorBackLinked @RT(0) @T @F @DT @RT(4)BOOL @RT(0) @T @T @BASIC 0 @F
@F @F
@T
@BEG_Attrib
3 @RT(0) @RT(0) @RT(0)
@END_Attrib
1 0 @F @F @F @F

@Var @RT(13)fbEPUnForceAI @RT(0) @T @T @DERIVED 0 @T @T @DT @RT(13)FBEPUnForceAI @RT(0) @T @T @UNKNOWN 0 @F
@F @F
@T
@BEG_Attrib
3 @RT(0) @RT(0) @RT(0)
@END_Attrib
1 0 @F @F @F @F

@Var @RT(13)fbEPUnForceDI @RT(0) @T @T @DERIVED 0 @T @T @DT @RT(13)FBEPUnForceDI @RT(0) @T @T @UNKNOWN 0 @F
@F @F
@T
@BEG_Attrib
3 @RT(0) @RT(0) @RT(0)
@END_Attrib
1 0 @F @F @F @F

@Var @RT(10)TaskAnalog @RT(0) @T @T @RENAMED 0 @T @T @DT @RT(4)TASK @RT(0) @T @T @BASIC 0 @F
@F @F
@T
@BEG_Attrib
3 @RT(0) @RT(0) @RT(0)
@END_Attrib
1 7 @F @F @F @F

@Var @RT(19)sv_ForceEjectorBack @RT(0) @T @T @RENAMED 0 @T @T @DT @RT(4)BOOL @RT(0) @T @T @BASIC 0 @F
@F @F
@T
@BEG_Attrib
3 @RT(0) @RT(0) @RT(0)
@END_Attrib
1 8 @F @F @F @F

@Var @RT(7)mpPumps @RT(0) @T @T @REFTO 0 @F @DERIVED 0 @T @T @DT @RT(15)tsRequiredPumps @RT(0) @T @T @UNKNOWN 0 @F
@F @F
@T
@BEG_Attrib
3 @RT(0) @RT(0) @RT(0)
@END_Attrib
1 0 @F @F @F @F

@Var @RT(12)sv_bInitDone @RT(0) @T @T @RENAMED 0 @T @T @DT @RT(4)BOOL @RT(0) @T @T @BASIC 0 @F
@F @F
@T
@BEG_Attrib
3 @RT(0) @RT(0) @RT(0)
@END_Attrib
1 8 @F @F @F @F

@Var @RT(11)mprVelocity @RT(0) @T @T @REFTO 0 @T @DT @RT(4)REAL @RT(0) @T @T @BASIC 0 @F
@F @F
@T
@BEG_Attrib
3 @RT(0) @RT(0) @RT(0)
@END_Attrib
1 0 @F @F @F @F

@Var @RT(21)fbGetSimulationSource @RT(0) @T @T @DERIVED 0 @T @T @DT @RT(21)FBGetSimulationSource @RT(0) @T @T @UNKNOWN 0 @F
@F @F
@T
@BEG_Attrib
3 @RT(0) @RT(0) @RT(0)
@END_Attrib
1 0 @F @F @F @F

@END_Dcl

@END_Export

@BEG_Body

6

@BEG_Export

@BEG_Algo
@POSTUPDATE_ALGORITHM @RT(6)pStart @STRUCTURED_TEXT
@RT(0) @RT(26)sv_bSimulate,sv_bInitStart @RT(10)PU_Task_13 @F @F
@END_Algo

@BEG_Dcl
@RT(16)DclTreeContainer
0
@END_Dcl

@END_Export

@BEG_Export

@BEG_Algo
@PROCESS_ALGORITHM @RT(10)paSimulate @SEQUENTIAL_FLOW_CHART
@RT(0) @RT(0) @RT(10)TaskAnalog @F @F
@END_Algo

@BEG_Dcl
@RT(16)DclTreeContainer
17
@Var @RT(14)rEjectDivision @RT(0) @T @F @DT @RT(4)REAL @RT(0) @T @T @BASIC 0 @F
@F @F
@T
@BEG_Attrib
3 @RT(3)0.3 @RT(0) @RT(0)
@END_Attrib
1 0 @F @F @F @F

@Var @RT(15)mrEjectorPosRaw @RT(0) @T @F @DT @RT(4)REAL @RT(0) @T @T @BASIC 0 @F
@F @F
@T
@BEG_Attrib
3 @RT(0) @RT(0) @RT(0)
@END_Attrib
1 0 @F @F @F @F

@Var @RT(16)rEjectTimeFor10V @RT(0) @T @F @DT @RT(4)REAL @RT(0) @T @T @BASIC 0 @F
@F @F
@T
@BEG_Attrib
3 @RT(3)1.0 @RT(0) @RT(0)
@END_Attrib
1 0 @F @F @F @F

@Var @RT(8)TimerFwd @RT(0) @T @T @DERIVED 0 @T @T @DT @RT(3)TON @RT(0) @T @T @UNKNOWN 0 @F
@F @F
@T
@BEG_Attrib
3 @RT(0) @RT(16)chad(CR_0038565) @RT(0)
@END_Attrib
1 0 @F @F @F @F

@Var @RT(8)TimerBwd @RT(0) @T @T @DERIVED 0 @T @T @DT @RT(3)TON @RT(0) @T @T @UNKNOWN 0 @F
@F @F
@T
@BEG_Attrib
3 @RT(0) @RT(16)chad(CR_0038565) @RT(0)
@END_Attrib
1 0 @F @F @F @F

@Var @RT(10)rCycleTime @RT(0) @T @F @DT @RT(4)REAL @RT(0) @T @T @BASIC 0 @F
@F @F
@T
@BEG_Attrib
3 @RT(0) @RT(0) @RT(0)
@END_Attrib
1 0 @F @F @F @F

@Var @RT(10)dCycleTime @RT(0) @T @F @DT @RT(4)TIME @RT(0) @T @T @BASIC 0 @F
@F @F
@T
@BEG_Attrib
3 @RT(0) @RT(0) @RT(0)
@END_Attrib
1 0 @F @F @F @F

@Var @RT(15)prEjectorPosRaw @RT(0) @T @T @REFTO 0 @T @DT @RT(4)REAL @RT(0) @T @T @BASIC 0 @F
@F @F
@T
@BEG_Attrib
3 @RT(0) @RT(0) @RT(0)
@END_Attrib
1 0 @F @F @F @F

@Var @RT(21)bAIEjectorTransLinked @RT(0) @T @F @DT @RT(4)BOOL @RT(0) @T @T @BASIC 0 @F
@F @F
@T
@BEG_Attrib
3 @RT(0) @RT(0) @RT(0)
@END_Attrib
1 0 @F @F @F @F

@Var @RT(14)pbDOEjectorBwd @RT(0) @T @T @REFTO 0 @T @DT @RT(4)BOOL @RT(0) @T @T @BASIC 0 @F
@F @F
@T
@BEG_Attrib
3 @RT(0) @RT(0) @RT(0)
@END_Attrib
1 0 @F @F @F @F

@Var @RT(14)pbDOEjectorFwd @RT(0) @T @T @REFTO 0 @T @DT @RT(4)BOOL @RT(0) @T @T @BASIC 0 @F
@F @F
@T
@BEG_Attrib
3 @RT(0) @RT(0) @RT(0)
@END_Attrib
1 0 @F @F @F @F

@Var @RT(19)bDOEjectorFwdLinked @RT(0) @T @F @DT @RT(4)BOOL @RT(0) @T @T @BASIC 0 @F
@F @F
@T
@BEG_Attrib
3 @RT(0) @RT(0) @RT(0)
@END_Attrib
1 0 @F @F @F @F

@Var @RT(19)bDOEjectorBwdLinked @RT(0) @T @F @DT @RT(4)BOOL @RT(0) @T @T @BASIC 0 @F
@F @F
@T
@BEG_Attrib
3 @RT(0) @RT(0) @RT(0)
@END_Attrib
1 0 @F @F @F @F

@Var @RT(19)bDIEjectorFwdLinked @RT(0) @T @F @DT @RT(4)BOOL @RT(0) @T @T @BASIC 0 @F
@F @F
@T
@BEG_Attrib
3 @RT(0) @RT(16)chad(CR_0038565) @RT(0)
@END_Attrib
1 0 @F @F @F @F

@Var @RT(7)pbDummy @RT(0) @T @T @REFTO 0 @T @DT @RT(4)BOOL @RT(0) @T @T @BASIC 0 @F
@F @F
@T
@BEG_Attrib
3 @RT(0) @RT(0) @RT(0)
@END_Attrib
1 0 @F @F @F @F

@Var @RT(6)Status @RT(0) @T @T @DERIVED 0 @T @T @DT @RT(11)KSYS_Status @RT(0) @T @T @UNKNOWN 0 @F
@F @F
@T
@BEG_Attrib
3 @RT(0) @RT(0) @RT(0)
@END_Attrib
1 0 @F @F @F @F

@Var @RT(27)bDIEjectorSafetyPlateLinked @RT(0) @T @F @DT @RT(4)BOOL @RT(0) @T @T @BASIC 0 @F
@F @F
@T
@BEG_Attrib
3 @RT(0) @RT(0) @RT(0)
@END_Attrib
1 0 @F @F @F @F

@END_Dcl

@END_Export

@BEG_Export

@BEG_Algo
@POSTUPDATE_ALGORITHM @RT(11)pEjectorBwd @STRUCTURED_TEXT
@RT(0) @RT(19)sv_ForceEjectorBack @RT(7)TaskSim @F @F
@END_Algo

@BEG_Dcl
@RT(16)DclTreeContainer
0
@END_Dcl

@END_Export

@BEG_Export

@BEG_Algo
@ALGORITHM @RT(20)aGetSimulationSource @STRUCTURED_TEXT
@RT(0) @RT(0) @RT(0) @F @F
@END_Algo

@BEG_Dcl
@RT(16)DclTreeContainer
0
@END_Dcl

@END_Export

@BEG_Export

@BEG_Algo
@POSTUPDATE_ALGORITHM @RT(9)pInitDone @STRUCTURED_TEXT
@RT(0) @RT(12)sv_bInitDone @RT(7)TaskSim @F @F
@END_Algo

@BEG_Dcl
@RT(16)DclTreeContainer
1
@Var @RT(18)fbGetRequiredPumps @RT(0) @T @T @DERIVED 0 @T @T @DT @RT(18)FBGetRequiredPumps @RT(0) @T @T @UNKNOWN 0 @F
@F @F
@T
@BEG_Attrib
3 @RT(0) @RT(0) @RT(0)
@END_Attrib
1 0 @F @F @F @F

@END_Dcl

@END_Export

@BEG_Export

@BEG_Algo
@POSTUPDATE_ALGORITHM @RT(14)pRequiredPumps @STRUCTURED_TEXT
@RT(0) @RT(22)mpPumps^.RequiredPumps @RT(7)TaskSim @F @F
@END_Algo

@BEG_Dcl
@RT(16)DclTreeContainer
0
@END_Dcl

@END_Export

@BEG_Body
@TL(9)
(**************************************** WARNING ********************************************
 *** The KEBA Kemro K2 System including software is not intended for safety control tasks! ***
 ***                       For further information see Comment tab!                        ***
 *********************************************************************************************)

IF sv_bSimulate THEN
   START_PROCESS_ALGORITHM(paSimulate);
END_IF;

@END_Body

@@@BEG_Comment@@@
@TL(0)

@@@END_Comment@@@

@BEG_SfcBody
4 4 4

@BEG_SfcData 2
@StepSeq @RT(4)sseq @F 3
@Step @RT(4)INIT @F @T @F @F @RT(0) @F
@AcbCont @RT(7)unnamed @F 1
@Acb @RT(5)aInit @F @F @RT(1)P @RT(0) @F @F @F @F

@Trans @RT(11)SimRequired @F @T @F @F @T @T @TL(2)
sv_bSimulate

@RT(11)SimRequired @F
@Loop @RT(4)loop @F 2
@StepSeq @RT(4)sseq @F 3
@Step @RT(3)SIM @F @F @F @F @RT(0) @F
@AcbCont @RT(7)unnamed @F 1
@Acb @RT(9)aSimulate @F @F @RT(1)N @RT(0) @F @F @F @F

@Trans @RT(14)StpSimRequired @F @T @F @F @T @T @TL(2)
NOT sv_bSimulate

@RT(14)StpSimRequired @F
@Step @RT(4)STOP @F @F @F @F @RT(0) @F
@AcbCont @RT(7)unnamed @F 1
@Acb @RT(9)aStopSimu @F @F @RT(1)P @RT(0) @F @F @F @F

@Trans @RT(6)Return @F @T @T @T @T @T @TL(2)
TRUE

@RT(6)Return @F

@END_SfcData
@SaActions 3
@SaText @RT(5)aInit 1 @TL(42)
(**************************************** WARNING ********************************************
 *** The KEBA Kemro K2 System including software is not intended for safety control tasks! ***
 ***                       For further information see Comment tab!                        ***
 *********************************************************************************************)

pbDummy := GET_SYNC_REFTO('Ejector1.di_EjectorBwd', T#0s, Status);
mbDIEjectorBackLinked := (Status = KSYS_Status_OK);

pbDummy := GET_SYNC_REFTO('Ejector1.di_EjectorFwd', T#0s, Status);
bDIEjectorFwdLinked := (Status = KSYS_Status_OK);

prEjectorPosRaw := GET_SYNC_REFTO('Ejector1.ai_Position', T#0s, Status);
bAIEjectorTransLinked := (Status = KSYS_Status_OK);

pbDOEjectorFwd := GET_SYNC_REFTO('Ejector1.do_Forward', T#0s, Status);
bDOEjectorFwdLinked := (Status = KSYS_Status_OK);

pbDOEjectorBwd := GET_SYNC_REFTO('Ejector1.do_Backward', T#0s, Status);
bDOEjectorBwdLinked := (Status = KSYS_Status_OK);

pbDummy := GET_SYNC_REFTO('Ejector1.di_SafetyPlate', T#0s, Status);
bDIEjectorSafetyPlateLinked := (Status = KSYS_Status_OK);
IF bDIEjectorSafetyPlateLinked THEN
   fbEPForceDI(sSysVar := 'Ejector1.di_SafetyPlate',Value := TRUE);
END_IF;

dCycleTime :=  GET_TASK_INTERVAL();
rCycleTime := (LINT_TO_REAL(TIME_TO_LINT(dCycleTime))) / 1000000.0;
rEjectDivision := 1.0  / rEjectTimeFor10V * rCycleTime;

sv_ForceEjectorBack := TRUE;

IF bDIEjectorFwdLinked THEN    //chad(CR_0038565)
   fbEPForceDI(sSysVar := 'Ejector1.di_EjectorFwd',Value := FALSE);
END_IF;

IF bAIEjectorTransLinked THEN
   ai_Position_stat := FALSE;
   fbEPForceAI(sSysVar := 'Ejector1.ai_Position',Value := 0.0, Range := 10.0);
END_IF;

@SaText @RT(9)aSimulate 1 @TL(56)
(**************************************** WARNING ********************************************
 *** The KEBA Kemro K2 System including software is not intended for safety control tasks! ***
 ***                       For further information see Comment tab!                        ***
 *********************************************************************************************)

IF bAIEjectorTransLinked THEN
   IF bDOEjectorFwdLinked AND pbDOEjectorFwd^ THEN
      mrEjectorPosRaw := prEjectorPosRaw^ + MUL(rEjectDivision,mprVelocity^);
      sv_ForceEjectorBack := FALSE;
   ELSIF bDOEjectorBwdLinked AND pbDOEjectorBwd^ THEN
      mrEjectorPosRaw := prEjectorPosRaw^ - MUL(rEjectDivision,mprVelocity^);
      IF prEjectorPosRaw^ <= 2.0 THEN
            sv_ForceEjectorBack := TRUE;
      END_IF;
   END_IF;
   fbEPForceAI(sSysVar := 'Ejector1.ai_Position', Value := MAX(mrEjectorPosRaw,0.0), Range := 10.0);

ELSE    //chad(CR_0038565) - transducer not linked

   //Move forward simulation
   IF bDOEjectorFwdLinked AND (NOT pbDOEjectorFwd^) THEN
      TimerFwd(IN := FALSE);
   END_IF;

   IF bDOEjectorFwdLinked AND pbDOEjectorFwd^ THEN
      TimerFwd(IN := TRUE, PT := t#4s);
      IF mbDIEjectorBackLinked THEN
         sv_ForceEjectorBack := FALSE;
         TimerBwd(IN := FALSE);
      END_IF;

      IF TimerFwd.Q AND bDIEjectorFwdLinked THEN
         fbEPForceDI(sSysVar := 'Ejector1.di_EjectorFwd',Value := TRUE);
         TimerFwd(IN := FALSE);
      END_IF;
   END_IF;

   //Move backward simulation
   IF bDOEjectorBwdLinked AND (NOT pbDOEjectorBwd^) THEN
      TimerBwd(IN := FALSE);
   END_IF;

   IF bDOEjectorBwdLinked AND pbDOEjectorBwd^ THEN
      TimerBwd(IN := TRUE, PT := t#4s);
      IF bDIEjectorFwdLinked THEN
         fbEPForceDI(sSysVar := 'Ejector1.di_EjectorFwd',Value := FALSE);
         TimerFwd(IN := FALSE);
      END_IF;

      IF TimerBwd.Q AND mbDIEjectorBackLinked THEN
         sv_ForceEjectorBack := TRUE;
         TimerBwd(IN := FALSE);
      END_IF;
   END_IF;
END_IF;

@SaText @RT(9)aStopSimu 1 @TL(20)
(**************************************** WARNING ********************************************
 *** The KEBA Kemro K2 System including software is not intended for safety control tasks! ***
 ***                       For further information see Comment tab!                        ***
 *********************************************************************************************)

IF bAIEjectorTransLinked THEN
   fbEPUnForceAI(sSysVar := 'Ejector1.ai_Position');
END_IF;
IF mbDIEjectorBackLinked THEN
   fbEPUnForceDI(sSysVar := 'Ejector1.di_EjectorBwd');
END_IF;
IF bDIEjectorSafetyPlateLinked THEN
   fbEPUnForceDI(sSysVar := 'Ejector1.di_SafetyPlate');
END_IF;
IF bDIEjectorFwdLinked THEN   //chad(CR_0038565)
   fbEPUnForceDI(sSysVar := 'Ejector1.di_EjectorFwd');
END_IF;

STOP_PROCESS_ALGORITHM();

@SaTrans 0
@SaExits 0
@END_SfcBody

@@@BEG_Comment@@@
@TL(0)

@@@END_Comment@@@

@BEG_Body
@TL(9)
(**************************************** WARNING ********************************************
 *** The KEBA Kemro K2 System including software is not intended for safety control tasks! ***
 ***                       For further information see Comment tab!                        ***
 *********************************************************************************************)

IF mbDIEjectorBackLinked THEN
   fbEPForceDI(sSysVar := 'Ejector1.di_EjectorBwd',Value := sv_ForceEjectorBack);
END_IF;

@END_Body

@@@BEG_Comment@@@
@TL(0)

@@@END_Comment@@@

@BEG_Body
@TL(8)
(**************************************** WARNING ********************************************
 *** The KEBA Kemro K2 System including software is not intended for safety control tasks! ***
 ***                       For further information see Comment tab!                        ***
 *********************************************************************************************)

fbGetSimulationSource(pRequiredPumps := mpPumps,
                      prVelocity => mprVelocity);

@END_Body

@@@BEG_Comment@@@
@TL(0)

@@@END_Comment@@@

@BEG_Body
@TL(17)
(**************************************** WARNING ********************************************
 *** The KEBA Kemro K2 System including software is not intended for safety control tasks! ***
 ***                       For further information see Comment tab!                        ***
 *********************************************************************************************)

//get required pumps
fbGetRequiredPumps.DeviceId.CompId := cCompEjector;
fbGetRequiredPumps.DeviceId.IndexId := 1;

fbGetRequiredPumps(MoveDir := cMoveFwd,
                   MoveId := cMoveFwd);
mpPumps := fbGetRequiredPumps.pPumps;

aGetSimulationSource();

@END_Body

@@@BEG_Comment@@@
@TL(0)

@@@END_Comment@@@

@BEG_Body
@TL(7)
(**************************************** WARNING ********************************************
 *** The KEBA Kemro K2 System including software is not intended for safety control tasks! ***
 ***                       For further information see Comment tab!                        ***
 *********************************************************************************************)

aGetSimulationSource();

@END_Body

@@@BEG_Comment@@@
@TL(0)

@@@END_Comment@@@
@END_Body

@END_Contents

(* ---- ABEnergyMeterSimu.pu ---- *)
IMPORT_OVER_LISTFILE
 GET_SYNC_REFTO
, cApplPlasticsPI
, cCompEnergyMeter
, cSubOpSpeedpumpMaster
, tyNumberOfDevices
, KSYS_Status
, tOptionId
, KSWO_Status

END_IMPORT

ALGORITHM_BLOCK ABEnergyMeterSimu #DUMMY_EDIT_BLOCK

SYSTEM_VAR
 sv_bSimulate : BOOL;
 sv_bInitStart : BOOL;
 sv_NumberOfDevices : tyNumberOfDevices;
 sv_rMeasuredPower : REAL;
 sv_rMeasuredEnergy : REAL;
 sv_rHeatingPower : REAL;
 sv_rIdlePower : REAL;
END_VAR

SYSTEM_OBJECT
 TaskSim : TASK;
 TaskSlow : TASK;
 TaskInject : TASK;
 TaskAnalog : TASK;
END_OBJECT

VAR
 mbEnergyMeterLinked : BOOL;
 mbSpeedPump : BOOL;
 mprMotorTotalPower : REFTO REAL;
END_VAR

PROCESS_ALGORITHM paSimulate ON TaskAnalog

VAR_TEMP
 b : BOOL;
END_VAR

VAR
 Status : KSYS_Status;
 dCycleTime : TIME;
 rCycleTime : REAL;
 rInitialEnergy : REAL := 500000.0;
 rMotorPower : REAL := 20000.0;
 rOldMeasuredEnergy : REAL;
 rMeasuredPower : REAL := 20000.0;
END_VAR

(* IecGraph-Code *)

(* init step *)
INITIAL_STEP INIT:
aInit (P);
END_STEP

(* steps *)
STEP SIM:
aSimulate (N);
END_STEP

STEP STOP:
aStopSimu (P);
END_STEP

(* transitions *)
TRANSITION SimRequired (* SimRequired *) FROM INIT TO SIM :=  #BEGIN_EDIT_BLOCK
sv_bSimulate
;#END_EDIT_BLOCK
END_TRANSITION

TRANSITION StpSimRequired (* StpSimRequired *) FROM SIM TO STOP :=  #BEGIN_EDIT_BLOCK
NOT sv_bSimulate
;#END_EDIT_BLOCK
END_TRANSITION

TRANSITION Return (* Return *) FROM STOP TO SIM :=  #BEGIN_EDIT_BLOCK
TRUE
;#END_EDIT_BLOCK
END_TRANSITION

(* end IecGraph-Code *)
(* sfc-code *)

(* stand alone actions *)
ACTION aInit: #BEGIN_EDIT_BLOCK
(**************************************** WARNING ********************************************
 *** The KEBA Kemro K2 System including software is not intended for safety control tasks! ***
 ***                       For further information see Comment tab!                        ***
 *********************************************************************************************)

//Use motor simulation in case of speedpump
IF mbSpeedPump THEN
   mprMotorTotalPower := GET_SYNC_REFTO('Pump1.sv_rMotorTotalPower', T#0s, Status);
END_IF;

dCycleTime := GET_TASK_INTERVAL();
rCycleTime := (LINT_TO_REAL(TIME_TO_LINT(dCycleTime))) / 1000000.0;

b := WRITE_SVREAL_DIRECT(sv_rMeasuredEnergy, rInitialEnergy);

;#END_EDIT_BLOCK END_ACTION (*aInit*)
ACTION aStopSimu: #BEGIN_EDIT_BLOCK
(**************************************** WARNING ********************************************
 *** The KEBA Kemro K2 System including software is not intended for safety control tasks! ***
 ***                       For further information see Comment tab!                        ***
 *********************************************************************************************)

STOP_PROCESS_ALGORITHM();

;#END_EDIT_BLOCK END_ACTION (*aStopSimu*)
ACTION aSimulate: #BEGIN_EDIT_BLOCK
(**************************************** WARNING ********************************************
 *** The KEBA Kemro K2 System including software is not intended for safety control tasks! ***
 ***                       For further information see Comment tab!                        ***
 *********************************************************************************************)

IF mbSpeedPump THEN
   rMotorPower := mprMotorTotalPower^ * 1.0e3;
   b := WRITE_SVREAL_DIRECT(sv_rMeasuredPower, (rMotorPower + sv_rHeatingPower + sv_rIdlePower)); //W
ELSE
   b := WRITE_SVREAL_DIRECT(sv_rMeasuredPower, rMeasuredPower);  //no speedpump
END_IF;

b := WRITE_SVREAL_DIRECT(sv_rMeasuredEnergy, (sv_rMeasuredPower * rCycleTime / 3600.0 + rOldMeasuredEnergy)); //Wh
rOldMeasuredEnergy := sv_rMeasuredEnergy;

;#END_EDIT_BLOCK END_ACTION (*aSimulate*)
(* end sfc-code *)

END_ALGORITHM

POSTUPDATE_ALGORITHM pStart ON TaskSim WITH sv_bSimulate,sv_bInitStart

VAR
 bInitDone : BOOL;
 pOptions : REFTO tOptionId;
 s : KSYS_Status;
END_VAR
#BEGIN_EDIT_BLOCK
(**************************************** WARNING ********************************************
 *** The KEBA Kemro K2 System including software is not intended for safety control tasks! ***
 ***                       For further information see Comment tab!                        ***
 *********************************************************************************************)

IF NOT bInitDone THEN
   //check if the energy meter is linked
   IF sv_NumberOfDevices[cCompEnergyMeter] <> 0 THEN
      mbEnergyMeterLinked := TRUE;
   END_IF;

   pOptions := GET_SYNC_REFTO('Pump1.sv_Options', T#0s, s);
   mbSpeedPump := (s = KSYS_Status_OK) AND ((pOptions^ AND cSubOpSpeedpumpMaster) = cSubOpSpeedpumpMaster);
   bInitDone := TRUE;
END_IF;

IF sv_bSimulate AND mbEnergyMeterLinked THEN
   START_PROCESS_ALGORITHM(paSimulate);
END_IF;

;#END_EDIT_BLOCK END_ALGORITHM

PROCESS_ALGORITHM paInitDebugMeasurement ON TaskSlow AUTOSTART

VAR
 fuName : STRING(255);
 variableName : STRING(255);
 swoState : KSWO_Status;
END_VAR
#BEGIN_EDIT_BLOCK
(**************************************** WARNING ********************************************
 *** The KEBA Kemro K2 System including software is not intended for safety control tasks! ***
 ***                       For further information see Comment tab!                        ***
 *********************************************************************************************)

fuName := GET_MY_FU_NAME();
variableName := CONCAT(fuName,'.rMeasuredPower kW');
swoState := KSWO_AddVariable( Task := TaskInject,
                              Name := variableName,
                              Variable := sv_rMeasuredPower);

variableName := CONCAT(fuName,'.rMeasuredEnergy kWh');
swoState := KSWO_AddVariable( Task := TaskInject,
                              Name := variableName,
                              Variable := sv_rMeasuredEnergy);
STOP_PROCESS_ALGORITHM();

;#END_EDIT_BLOCK END_ALGORITHM

END_ALGORITHM_BLOCK

#END_OF_IEC_PART

@Puma @IecEditor 6 127 @Pou 25
@@@BEG_Comment@@@

@@@END_Comment@@@

@BEG_Contents

@BEG_Func
@RT(17)FuncTreeContainer
1
@Var @RT(14)GET_SYNC_REFTO @RT(0) @T @T @DERIVED 0 @F @RT(22)KEBA_STANDARD_FUNCTION @F
@T
@BEG_Attrib
0 @RT(0) @RT(0)
@END_Attrib
1 1 @F @F @F @F

@END_Func

@BEG_Const
@RT(18)ConstTreeContainer
3
@Var @RT(15)cApplPlasticsPI @RT(0) @T @F @DT @RT(4)REAL @RT(0) @T @T @BASIC 0 @F
@F @F
@T
@BEG_Attrib
0 @RT(10)3.14159265 @RT(13)pi=3.14159265
@END_Attrib
1 1 @F @F @F @F

@Var @RT(16)cCompEnergyMeter @RT(0) @T @F @DT @RT(4)DINT @RT(0) @T @T @BASIC 0 @F
@F @F
@T
@BEG_Attrib
0 @RT(3)157 @RT(22)Component Energy meter
@END_Attrib
1 1 @F @F @F @F

@Var @RT(21)cSubOpSpeedpumpMaster @RT(0) @T @F @DT @RT(5)DWORD @RT(0) @T @T @BASIC 0 @F
@F @F
@T
@BEG_Attrib
0 @RT(6)16#100 @RT(17)Speed pump Master
@END_Attrib
1 1 @F @F @F @F

@END_Const

@BEG_Export

@BEG_Kind
@ALGORITHM_BLOCK @RT(17)ABEnergyMeterSimu @STRUCTURED_TEXT
@RT(0) @RT(0) @RT(0)
@END_Kind

@BEG_Dcl
@RT(16)DclTreeContainer
14
@Var @RT(7)TaskSim @RT(0) @T @F @DT @RT(4)TASK @RT(0) @T @T @BASIC 0 @F
@F @F
@T
@BEG_Attrib
3 @RT(0) @RT(0) @RT(0)
@END_Attrib
1 7 @F @F @F @F

@Var @RT(8)TaskSlow @RT(0) @T @F @DT @RT(4)TASK @RT(0) @T @T @BASIC 0 @F
@F @F
@T
@BEG_Attrib
3 @RT(0) @RT(0) @RT(0)
@END_Attrib
1 7 @F @F @F @F

@Var @RT(10)TaskInject @RT(0) @T @F @DT @RT(4)TASK @RT(0) @T @T @BASIC 0 @F
@F @F
@T
@BEG_Attrib
3 @RT(0) @RT(0) @RT(0)
@END_Attrib
1 7 @F @F @F @F

@Var @RT(10)TaskAnalog @RT(0) @T @T @RENAMED 0 @T @T @DT @RT(4)TASK @RT(0) @T @T @BASIC 0 @F
@F @F
@T
@BEG_Attrib
3 @RT(0) @RT(0) @RT(0)
@END_Attrib
1 7 @F @F @F @F

@Var @RT(12)sv_bSimulate @RT(0) @T @F @DT @RT(4)BOOL @RT(0) @T @T @BASIC 0 @F
@F @F
@T
@BEG_Attrib
3 @RT(0) @RT(0) @RT(0)
@END_Attrib
1 8 @F @F @F @F

@Var @RT(13)sv_bInitStart @RT(0) @T @F @DT @RT(4)BOOL @RT(0) @T @T @BASIC 0 @F
@F @F
@T
@BEG_Attrib
3 @RT(0) @RT(0) @RT(0)
@END_Attrib
1 8 @F @F @F @F

@Var @RT(18)sv_NumberOfDevices @RT(0) @T @T @DERIVED 0 @T @T @DT @RT(17)tyNumberOfDevices @RT(0) @T @T @UNKNOWN 0 @F
@F @F
@T
@BEG_Attrib
3 @RT(0) @RT(0) @RT(0)
@END_Attrib
1 8 @F @F @F @F

@Var @RT(19)mbEnergyMeterLinked @RT(0) @T @T @RENAMED 0 @T @T @DT @RT(4)BOOL @RT(0) @T @T @BASIC 0 @F
@F @F
@T
@BEG_Attrib
3 @RT(0) @RT(0) @RT(0)
@END_Attrib
1 0 @F @F @F @F

@Var @RT(17)sv_rMeasuredPower @RT(0) @T @F @DT @RT(4)REAL @RT(0) @T @T @BASIC 0 @F
@F @F
@T
@BEG_Attrib
3 @RT(0) @RT(0) @RT(0)
@END_Attrib
1 8 @F @F @F @F

@Var @RT(18)sv_rMeasuredEnergy @RT(0) @T @F @DT @RT(4)REAL @RT(0) @T @T @BASIC 0 @F
@F @F
@T
@BEG_Attrib
3 @RT(0) @RT(0) @RT(0)
@END_Attrib
1 8 @F @F @F @F

@Var @RT(16)sv_rHeatingPower @RT(0) @T @F @DT @RT(4)REAL @RT(0) @T @T @BASIC 0 @F
@F @F
@T
@BEG_Attrib
3 @RT(0) @RT(0) @RT(0)
@END_Attrib
1 8 @F @F @F @F

@Var @RT(13)sv_rIdlePower @RT(0) @T @F @DT @RT(4)REAL @RT(0) @T @T @BASIC 0 @F
@F @F
@T
@BEG_Attrib
3 @RT(0) @RT(0) @RT(0)
@END_Attrib
1 8 @F @F @F @F

@Var @RT(11)mbSpeedPump @RT(0) @T @T @RENAMED 0 @T @T @DT @RT(4)BOOL @RT(0) @T @T @BASIC 0 @F
@F @F
@T
@BEG_Attrib
3 @RT(0) @RT(0) @RT(0)
@END_Attrib
1 0 @F @F @F @F

@Var @RT(18)mprMotorTotalPower @RT(0) @T @T @REFTO 0 @T @DT @RT(4)REAL @RT(0) @T @T @BASIC 0 @F
@F @F
@T
@BEG_Attrib
3 @RT(0) @RT(0) @RT(0)
@END_Attrib
1 0 @F @F @F @F

@END_Dcl

@END_Export

@BEG_Body

3

@BEG_Export

@BEG_Algo
@PROCESS_ALGORITHM @RT(10)paSimulate @SEQUENTIAL_FLOW_CHART
@RT(0) @RT(0) @RT(10)TaskAnalog @F @F
@END_Algo

@BEG_Dcl
@RT(16)DclTreeContainer
8
@Var @RT(6)Status @RT(0) @T @T @DERIVED 0 @T @T @DT @RT(11)KSYS_Status @RT(0) @T @T @UNKNOWN 0 @F
@F @F
@T
@BEG_Attrib
3 @RT(0) @RT(0) @RT(0)
@END_Attrib
1 0 @F @F @F @F

@Var @RT(10)dCycleTime @RT(0) @T @T @RENAMED 0 @T @T @DT @RT(4)TIME @RT(0) @T @T @BASIC 0 @F
@F @F
@T
@BEG_Attrib
3 @RT(0) @RT(0) @RT(0)
@END_Attrib
1 0 @F @F @F @F

@Var @RT(10)rCycleTime @RT(0) @T @F @DT @RT(4)REAL @RT(0) @T @T @BASIC 0 @F
@F @F
@T
@BEG_Attrib
3 @RT(0) @RT(0) @RT(0)
@END_Attrib
1 0 @F @F @F @F

@Var @RT(14)rInitialEnergy @RT(0) @T @T @RENAMED 0 @T @T @DT @RT(4)REAL @RT(0) @T @T @BASIC 0 @F
@F @F
@T
@BEG_Attrib
3 @RT(8)500000.0 @RT(0) @RT(0)
@END_Attrib
1 0 @F @F @F @F

@Var @RT(11)rMotorPower @RT(0) @T @T @RENAMED 0 @T @T @DT @RT(4)REAL @RT(0) @T @T @BASIC 0 @F
@F @F
@T
@BEG_Attrib
3 @RT(7)20000.0 @RT(0) @RT(0)
@END_Attrib
1 0 @F @F @F @F

@Var @RT(18)rOldMeasuredEnergy @RT(0) @T @T @RENAMED 0 @T @T @DT @RT(4)REAL @RT(0) @T @T @BASIC 0 @F
@F @F
@T
@BEG_Attrib
3 @RT(0) @RT(0) @RT(0)
@END_Attrib
1 0 @F @F @F @F

@Var @RT(14)rMeasuredPower @RT(0) @T @T @RENAMED 0 @T @T @DT @RT(4)REAL @RT(0) @T @T @BASIC 0 @F
@F @F
@T
@BEG_Attrib
3 @RT(7)20000.0 @RT(0) @RT(0)
@END_Attrib
1 0 @F @F @F @F

@Var @RT(1)b @RT(0) @T @F @DT @RT(4)BOOL @RT(0) @T @T @BASIC 0 @F
@F @F
@T
@BEG_Attrib
3 @RT(0) @RT(0) @RT(0)
@END_Attrib
1 4 @F @F @F @F

@END_Dcl

@END_Export

@BEG_Export

@BEG_Algo
@POSTUPDATE_ALGORITHM @RT(6)pStart @STRUCTURED_TEXT
@RT(0) @RT(26)sv_bSimulate,sv_bInitStart @RT(7)TaskSim @F @F
@END_Algo

@BEG_Dcl
@RT(16)DclTreeContainer
3
@Var @RT(9)bInitDone @RT(0) @T @F @DT @RT(4)BOOL @RT(0) @T @T @BASIC 0 @F
@F @F
@T
@BEG_Attrib
3 @RT(0) @RT(0) @RT(0)
@END_Attrib
1 0 @F @F @F @F

@Var @RT(8)pOptions @RT(0) @T @T @REFTO 0 @F @DERIVED 0 @T @T @DT @RT(9)tOptionId @RT(0) @T @T @UNKNOWN 0 @F
@F @F
@T
@BEG_Attrib
3 @RT(0) @RT(0) @RT(0)
@END_Attrib
1 0 @F @F @F @F

@Var @RT(1)s @RT(0) @T @T @DERIVED 0 @T @T @DT @RT(11)KSYS_Status @RT(0) @T @T @UNKNOWN 0 @F
@F @F
@T
@BEG_Attrib
3 @RT(0) @RT(0) @RT(0)
@END_Attrib
1 0 @F @F @F @F

@END_Dcl

@END_Export

@BEG_Export

@BEG_Algo
@PROCESS_ALGORITHM @RT(22)paInitDebugMeasurement @STRUCTURED_TEXT
@RT(0) @RT(0) @RT(8)TaskSlow @T @F
@END_Algo

@BEG_Dcl
@RT(16)DclTreeContainer
3
@Var @RT(6)fuName @RT(0) @T @F @DT @RT(11)STRING(255) @RT(0) @T @T @STRING 0 @F @RT(3)255 @F
@F @F
@T
@BEG_Attrib
3 @RT(0) @RT(0) @RT(0)
@END_Attrib
1 0 @F @F @F @F

@Var @RT(12)variableName @RT(0) @T @F @DT @RT(11)STRING(255) @RT(0) @T @T @STRING 0 @F @RT(3)255 @F
@F @F
@T
@BEG_Attrib
3 @RT(0) @RT(0) @RT(0)
@END_Attrib
1 0 @F @F @F @F

@Var @RT(8)swoState @RT(0) @T @T @DERIVED 0 @T @T @DT @RT(11)KSWO_Status @RT(0) @T @T @UNKNOWN 0 @F
@F @F
@T
@BEG_Attrib
3 @RT(0) @RT(0) @RT(0)
@END_Attrib
1 0 @F @F @F @F

@END_Dcl

@END_Export

@BEG_SfcBody
4 3 2

@BEG_SfcData 2
@StepSeq @RT(4)sseq @F 3
@Step @RT(4)INIT @F @T @F @F @RT(0) @F
@AcbCont @RT(7)unnamed @F 1
@Acb @RT(5)aInit @F @F @RT(1)P @RT(0) @F @F @F @F

@Trans @RT(11)SimRequired @F @T @F @F @T @T @TL(2)
sv_bSimulate

@RT(11)SimRequired @F
@Loop @RT(4)loop @F 2
@StepSeq @RT(4)sseq @F 3
@Step @RT(3)SIM @F @F @F @F @RT(0) @F
@AcbCont @RT(7)unnamed @F 1
@Acb @RT(9)aSimulate @F @F @RT(1)N @RT(0) @F @F @F @F

@Trans @RT(14)StpSimRequired @F @T @F @F @T @T @TL(2)
NOT sv_bSimulate

@RT(14)StpSimRequired @F
@Step @RT(4)STOP @F @F @F @F @RT(0) @F
@AcbCont @RT(7)unnamed @F 1
@Acb @RT(9)aStopSimu @F @F @RT(1)P @RT(0) @F @F @F @F

@Trans @RT(6)Return @F @T @T @T @T @T @TL(2)
TRUE

@RT(6)Return @F

@END_SfcData
@SaActions 3
@SaText @RT(5)aInit 1 @TL(15)
(**************************************** WARNING ********************************************
 *** The KEBA Kemro K2 System including software is not intended for safety control tasks! ***
 ***                       For further information see Comment tab!                        ***
 *********************************************************************************************)

//Use motor simulation in case of speedpump
IF mbSpeedPump THEN
   mprMotorTotalPower := GET_SYNC_REFTO('Pump1.sv_rMotorTotalPower', T#0s, Status);
END_IF;

dCycleTime := GET_TASK_INTERVAL();
rCycleTime := (LINT_TO_REAL(TIME_TO_LINT(dCycleTime))) / 1000000.0;

b := WRITE_SVREAL_DIRECT(sv_rMeasuredEnergy, rInitialEnergy);

@SaText @RT(9)aStopSimu 1 @TL(7)
(**************************************** WARNING ********************************************
 *** The KEBA Kemro K2 System including software is not intended for safety control tasks! ***
 ***                       For further information see Comment tab!                        ***
 *********************************************************************************************)

STOP_PROCESS_ALGORITHM();

@SaText @RT(9)aSimulate 1 @TL(17)
(**************************************** WARNING ********************************************
 *** The KEBA Kemro K2 System including software is not intended for safety control tasks! ***
 ***                       For further information see Comment tab!                        ***
 *********************************************************************************************)

IF mbSpeedPump THEN
   rMotorPower := mprMotorTotalPower^ * 1.0e3;
   b := WRITE_SVREAL_DIRECT(sv_rMeasuredPower, (rMotorPower + sv_rHeatingPower + sv_rIdlePower)); //W
ELSE
   b := WRITE_SVREAL_DIRECT(sv_rMeasuredPower, rMeasuredPower);  //no speedpump
END_IF;

b := WRITE_SVREAL_DIRECT(sv_rMeasuredEnergy, (sv_rMeasuredPower * rCycleTime / 3600.0 + rOldMeasuredEnergy)); //Wh
rOldMeasuredEnergy := sv_rMeasuredEnergy;

@SaTrans 0
@SaExits 0
@END_SfcBody

@@@BEG_Comment@@@
@TL(0)

@@@END_Comment@@@

@BEG_Body
@TL(20)
(**************************************** WARNING ********************************************
 *** The KEBA Kemro K2 System including software is not intended for safety control tasks! ***
 ***                       For further information see Comment tab!                        ***
 *********************************************************************************************)

IF NOT bInitDone THEN
   //check if the energy meter is linked
   IF sv_NumberOfDevices[cCompEnergyMeter] <> 0 THEN
      mbEnergyMeterLinked := TRUE;
   END_IF;

   pOptions := GET_SYNC_REFTO('Pump1.sv_Options', T#0s, s);
   mbSpeedPump := (s = KSYS_Status_OK) AND ((pOptions^ AND cSubOpSpeedpumpMaster) = cSubOpSpeedpumpMaster);
   bInitDone := TRUE;
END_IF;

IF sv_bSimulate AND mbEnergyMeterLinked THEN
   START_PROCESS_ALGORITHM(paSimulate);
END_IF;

@END_Body

@@@BEG_Comment@@@
@TL(0)

@@@END_Comment@@@

@BEG_Body
@TL(18)
(**************************************** WARNING ********************************************
 *** The KEBA Kemro K2 System including software is not intended for safety control tasks! ***
 ***                       For further information see Comment tab!                        ***
 *********************************************************************************************)

fuName := GET_MY_FU_NAME();
variableName := CONCAT(fuName,'.rMeasuredPower kW');
swoState := KSWO_AddVariable( Task := TaskInject,
                              Name := variableName,
                              Variable := sv_rMeasuredPower);

variableName := CONCAT(fuName,'.rMeasuredEnergy kWh');
swoState := KSWO_AddVariable( Task := TaskInject,
                              Name := variableName,
                              Variable := sv_rMeasuredEnergy);
STOP_PROCESS_ALGORITHM();

@END_Body

@@@BEG_Comment@@@
@TL(0)

@@@END_Comment@@@
@END_Body

@END_Contents

(* ---- ABEuromapSimulation.pu ---- *)
IMPORT_OVER_LISTFILE
 STOP_PROCESS_ALGORITHM
, CHECK_REF
, ABForceDigital

END_IMPORT

ALGORITHM_BLOCK ABEuromapSimulation #DUMMY_EDIT_BLOCK

SYSTEM_VAR
 sv_bSimulate : BOOL;
 sv_bInitStart : BOOL;
 sv_bRobotEmergencyStop : BOOL;
 sv_bRobotTurnedOn : BOOL;
END_VAR

SYSTEM_OBJECT
 PU_Task_7 : TASK;
 TaskSim : TASK;
END_OBJECT

VAR
 mbWantCleanup : BOOL;
 mbWantInit : BOOL;
 mbEnableEjectorBwd : BOOL := TRUE;
 mbEnableEjectorFwd : BOOL := TRUE;
 mbEnableCore1ToPos1 : BOOL := TRUE;
 mbEnableCore1ToPos2 : BOOL := TRUE;
 mbEnableCore2ToPos1 : BOOL := TRUE;
 mbEnableCore2ToPos2 : BOOL := TRUE;
 mbMoldAreaFree : BOOL := TRUE;
 mbEnableMoldClosure : BOOL := TRUE;
 mbEnableFullMoldOpening : BOOL := TRUE;
 abForceEmergencyStop : ABForceDigital;
 abForceRobotOperationMode : ABForceDigital;
 abForceRobotEnableEjectorFwd : ABForceDigital;
 abForceRobotEnableEjectorBwd : ABForceDigital;
 abForceRobotCore1ToPos1 : ABForceDigital;
 abForceRobotCore1ToPos2 : ABForceDigital;
 abForceRobotCore2ToPos1 : ABForceDigital;
 abForceRobotCore2ToPos2 : ABForceDigital;
 abForceRobotMoldAreaFree : ABForceDigital;
 abForceRobotEnableFullMoldOpen : ABForceDigital;
 abForceRobotEnableMoldClosure : ABForceDigital;
END_VAR

ALGORITHM aInit

VAR_OUTPUT
 bOK : BOOL;
END_VAR

VAR
 DeviceString : STRING(255);
END_VAR
#BEGIN_EDIT_BLOCK
mbWantInit := FALSE;
bOK := FALSE;
DeviceString := 'Euromap';

abForceEmergencyStop.aInit(Name := CONCAT(DeviceString, '.di_RobotEmergencyStop'));
abForceRobotOperationMode.aInit(Name := CONCAT(DeviceString, '.di_RobotOperationMode'));

abForceRobotEnableEjectorFwd.aInit(Name := CONCAT(DeviceString, '.di_EnableEjectorFwd'));
abForceRobotEnableEjectorBwd.aInit(Name := CONCAT(DeviceString, '.di_EnableEjectorBwd'));

abForceRobotCore1ToPos1.aInit(Name := CONCAT(DeviceString, '.di_EnableCore1ToPos1'));
abForceRobotCore1ToPos2.aInit(Name := CONCAT(DeviceString, '.di_EnableCore1ToPos2'));
abForceRobotCore2ToPos1.aInit(Name := CONCAT(DeviceString, '.di_EnableCore2ToPos1'));
abForceRobotCore2ToPos2.aInit(Name := CONCAT(DeviceString, '.di_EnableCore2ToPos2'));

abForceRobotMoldAreaFree.aInit(Name := CONCAT(DeviceString, '.di_MoldAreaFree'));
abForceRobotEnableFullMoldOpen.aInit(Name := CONCAT(DeviceString, '.di_EnableFullMoldOpening'));
abForceRobotEnableMoldClosure.aInit(Name := CONCAT(DeviceString, '.di_EnableMoldClosure'));

bOK := TRUE;

;#END_EDIT_BLOCK END_ALGORITHM

ALGORITHM aCleanup

#BEGIN_EDIT_BLOCK
mbWantCleanup := FALSE;

abForceEmergencyStop.aUnforce();
abForceRobotOperationMode.aUnforce();

abForceRobotEnableEjectorFwd.aUnforce();
abForceRobotEnableEjectorBwd.aUnforce();

abForceRobotCore1ToPos1.aUnforce();
abForceRobotCore1ToPos2.aUnforce();
abForceRobotCore2ToPos1.aUnforce();
abForceRobotCore2ToPos2.aUnforce();

abForceRobotMoldAreaFree.aUnforce();
abForceRobotEnableFullMoldOpen.aUnforce();
abForceRobotEnableMoldClosure.aUnforce();

;#END_EDIT_BLOCK END_ALGORITHM

POSTUPDATE_ALGORITHM pSimulateStart ON PU_Task_7 WITH sv_bSimulate,sv_bInitStart

#BEGIN_EDIT_BLOCK
IF sv_bSimulate THEN
   mbWantInit := TRUE;
   START_PROCESS_ALGORITHM(paSimulate);
ELSE
   mbWantCleanup := TRUE;
   START_PROCESS_ALGORITHM(paSimulate); //make sure it runs cleanup
END_IF;

;#END_EDIT_BLOCK END_ALGORITHM

PROCESS_ALGORITHM paSimulate ON TaskSim

#BEGIN_EDIT_BLOCK
IF mbWantInit THEN
   aInit();
   IF NOT aInit.bOK THEN
      STOP_PROCESS_ALGORITHM();
      RETURN;
   END_IF;
END_IF;

//TRUE = emergency stop OK
abForceEmergencyStop.aSetForceValue(bValue := NOT sv_bRobotEmergencyStop);

//FALSE = Operation with injection molding machine
//TRUE  = No operation with injection molding machine
abForceRobotOperationMode.aSetForceValue(bValue := NOT sv_bRobotTurnedOn);

//For now we just simulate that all movements are allowed immediately
abForceRobotEnableEjectorFwd.aSetForceValue(bValue := mbEnableEjectorFwd);
abForceRobotEnableEjectorBwd.aSetForceValue(bValue := mbEnableEjectorBwd);

abForceRobotCore1ToPos1.aSetForceValue(bValue := mbEnableCore1ToPos1);
abForceRobotCore1ToPos2.aSetForceValue(bValue := mbEnableCore1ToPos2);
abForceRobotCore2ToPos1.aSetForceValue(bValue := mbEnableCore2ToPos1);
abForceRobotCore2ToPos2.aSetForceValue(bValue := mbEnableCore2ToPos2);

abForceRobotMoldAreaFree.aSetForceValue(bValue := mbMoldAreaFree);
abForceRobotEnableFullMoldOpen.aSetForceValue(bValue := mbEnableMoldClosure);
abForceRobotEnableMoldClosure.aSetForceValue(bValue := mbEnableFullMoldOpening);

IF mbWantCleanup THEN
   aCleanup();
   STOP_PROCESS_ALGORITHM();
END_IF;

;#END_EDIT_BLOCK END_ALGORITHM

END_ALGORITHM_BLOCK

#END_OF_IEC_PART

@Puma @IecEditor 6 96 @Pou 25
@@@BEG_Comment@@@

@@@END_Comment@@@

@BEG_Contents

@BEG_Func
@RT(17)FuncTreeContainer
2
@Var @RT(22)STOP_PROCESS_ALGORITHM @RT(0) @T @T @DERIVED 0 @F @RT(23)KEBA_STANDARD_PROCEDURE @F
@T
@BEG_Attrib
0 @RT(0) @RT(0)
@END_Attrib
1 1 @F @F @F @F

@Var @RT(9)CHECK_REF @RT(0) @T @T @DERIVED 0 @F @RT(23)KEBA_STANDARD_PROCEDURE @F
@T
@BEG_Attrib
0 @RT(0) @RT(0)
@END_Attrib
1 1 @F @F @F @F

@END_Func

@BEG_Const
@RT(18)ConstTreeContainer
0
@END_Const

@BEG_Export

@BEG_Kind
@ALGORITHM_BLOCK @RT(19)ABEuromapSimulation @STRUCTURED_TEXT
@RT(0) @RT(0) @RT(0)
@END_Kind

@BEG_Dcl
@RT(16)DclTreeContainer
28
@Var @RT(9)PU_Task_7 @RT(0) @T @T @RENAMED 0 @T @T @DT @RT(4)TASK @RT(0) @T @T @BASIC 0 @F
@F @F
@T
@BEG_Attrib
3 @RT(0) @RT(0) @RT(0)
@END_Attrib
1 7 @F @F @F @F

@Var @RT(7)TaskSim @RT(0) @T @T @RENAMED 0 @T @T @DT @RT(4)TASK @RT(0) @T @T @BASIC 0 @F
@F @F
@T
@BEG_Attrib
3 @RT(0) @RT(0) @RT(0)
@END_Attrib
1 7 @F @F @F @F

@Var @RT(12)sv_bSimulate @RT(0) @T @T @RENAMED 0 @T @T @DT @RT(4)BOOL @RT(0) @T @T @BASIC 0 @F
@F @F
@T
@BEG_Attrib
3 @RT(0) @RT(0) @RT(0)
@END_Attrib
1 8 @F @F @F @F

@Var @RT(13)sv_bInitStart @RT(0) @T @F @DT @RT(4)BOOL @RT(0) @T @T @BASIC 0 @F
@F @F
@T
@BEG_Attrib
3 @RT(0) @RT(0) @RT(0)
@END_Attrib
1 8 @F @F @F @F

@Var @RT(22)sv_bRobotEmergencyStop @RT(0) @T @T @RENAMED 0 @T @T @DT @RT(4)BOOL @RT(0) @T @T @BASIC 0 @F
@F @F
@T
@BEG_Attrib
3 @RT(0) @RT(0) @RT(0)
@END_Attrib
1 8 @F @F @F @F

@Var @RT(17)sv_bRobotTurnedOn @RT(0) @T @T @RENAMED 0 @T @T @DT @RT(4)BOOL @RT(0) @T @T @BASIC 0 @F
@F @F
@T
@BEG_Attrib
3 @RT(0) @RT(0) @RT(0)
@END_Attrib
1 8 @F @F @F @F

@Var @RT(13)mbWantCleanup @RT(0) @T @F @DT @RT(4)BOOL @RT(0) @T @T @BASIC 0 @F
@F @F
@T
@BEG_Attrib
3 @RT(0) @RT(0) @RT(0)
@END_Attrib
1 0 @F @F @F @F

@Var @RT(10)mbWantInit @RT(0) @T @F @DT @RT(4)BOOL @RT(0) @T @T @BASIC 0 @F
@F @F
@T
@BEG_Attrib
3 @RT(0) @RT(0) @RT(0)
@END_Attrib
1 0 @F @F @F @F

@Var @RT(18)mbEnableEjectorBwd @RT(0) @T @F @DT @RT(4)BOOL @RT(0) @T @T @BASIC 0 @F
@F @F
@T
@BEG_Attrib
3 @RT(4)TRUE @RT(0) @RT(0)
@END_Attrib
1 0 @F @F @F @F

@Var @RT(18)mbEnableEjectorFwd @RT(0) @T @F @DT @RT(4)BOOL @RT(0) @T @T @BASIC 0 @F
@F @F
@T
@BEG_Attrib
3 @RT(4)TRUE @RT(0) @RT(0)
@END_Attrib
1 0 @F @F @F @F

@Var @RT(19)mbEnableCore1ToPos1 @RT(0) @T @F @DT @RT(4)BOOL @RT(0) @T @T @BASIC 0 @F
@F @F
@T
@BEG_Attrib
3 @RT(4)TRUE @RT(0) @RT(0)
@END_Attrib
1 0 @F @F @F @F

@Var @RT(19)mbEnableCore1ToPos2 @RT(0) @T @F @DT @RT(4)BOOL @RT(0) @T @T @BASIC 0 @F
@F @F
@T
@BEG_Attrib
3 @RT(4)TRUE @RT(0) @RT(0)
@END_Attrib
1 0 @F @F @F @F

@Var @RT(19)mbEnableCore2ToPos1 @RT(0) @T @F @DT @RT(4)BOOL @RT(0) @T @T @BASIC 0 @F
@F @F
@T
@BEG_Attrib
3 @RT(4)TRUE @RT(0) @RT(0)
@END_Attrib
1 0 @F @F @F @F

@Var @RT(19)mbEnableCore2ToPos2 @RT(0) @T @F @DT @RT(4)BOOL @RT(0) @T @T @BASIC 0 @F
@F @F
@T
@BEG_Attrib
3 @RT(4)TRUE @RT(0) @RT(0)
@END_Attrib
1 0 @F @F @F @F

@Var @RT(14)mbMoldAreaFree @RT(0) @T @F @DT @RT(4)BOOL @RT(0) @T @T @BASIC 0 @F
@F @F
@T
@BEG_Attrib
3 @RT(4)TRUE @RT(0) @RT(0)
@END_Attrib
1 0 @F @F @F @F

@Var @RT(19)mbEnableMoldClosure @RT(0) @T @F @DT @RT(4)BOOL @RT(0) @T @T @BASIC 0 @F
@F @F
@T
@BEG_Attrib
3 @RT(4)TRUE @RT(0) @RT(0)
@END_Attrib
1 0 @F @F @F @F

@Var @RT(23)mbEnableFullMoldOpening @RT(0) @T @F @DT @RT(4)BOOL @RT(0) @T @T @BASIC 0 @F
@F @F
@T
@BEG_Attrib
3 @RT(4)TRUE @RT(0) @RT(0)
@END_Attrib
1 0 @F @F @F @F

@Var @RT(20)abForceEmergencyStop @RT(0) @T @T @DERIVED 0 @T @T @DT @RT(14)ABForceDigital @RT(0) @T @T @UNKNOWN 0 @F
@F @F
@T
@BEG_Attrib
3 @RT(0) @RT(0) @RT(0)
@END_Attrib
1 0 @F @F @F @F

@Var @RT(25)abForceRobotOperationMode @RT(0) @T @T @DERIVED 0 @T @T @DT @RT(14)ABForceDigital @RT(0) @T @T @UNKNOWN 0 @F
@F @F
@T
@BEG_Attrib
3 @RT(0) @RT(0) @RT(0)
@END_Attrib
1 0 @F @F @F @F

@Var @RT(28)abForceRobotEnableEjectorFwd @RT(0) @T @T @DERIVED 0 @T @T @DT @RT(14)ABForceDigital @RT(0) @T @T @UNKNOWN 0 @F
@F @F
@T
@BEG_Attrib
3 @RT(0) @RT(0) @RT(0)
@END_Attrib
1 0 @F @F @F @F

@Var @RT(28)abForceRobotEnableEjectorBwd @RT(0) @T @T @DERIVED 0 @T @T @DT @RT(14)ABForceDigital @RT(0) @T @T @UNKNOWN 0 @F
@F @F
@T
@BEG_Attrib
3 @RT(0) @RT(0) @RT(0)
@END_Attrib
1 0 @F @F @F @F

@Var @RT(23)abForceRobotCore1ToPos1 @RT(0) @T @T @DERIVED 0 @T @T @DT @RT(14)ABForceDigital @RT(0) @T @T @UNKNOWN 0 @F
@F @F
@T
@BEG_Attrib
3 @RT(0) @RT(0) @RT(0)
@END_Attrib
1 0 @F @F @F @F

@Var @RT(23)abForceRobotCore1ToPos2 @RT(0) @T @T @DERIVED 0 @T @T @DT @RT(14)ABForceDigital @RT(0) @T @T @UNKNOWN 0 @F
@F @F
@T
@BEG_Attrib
3 @RT(0) @RT(0) @RT(0)
@END_Attrib
1 0 @F @F @F @F

@Var @RT(23)abForceRobotCore2ToPos1 @RT(0) @T @T @DERIVED 0 @T @T @DT @RT(14)ABForceDigital @RT(0) @T @T @UNKNOWN 0 @F
@F @F
@T
@BEG_Attrib
3 @RT(0) @RT(0) @RT(0)
@END_Attrib
1 0 @F @F @F @F

@Var @RT(23)abForceRobotCore2ToPos2 @RT(0) @T @T @DERIVED 0 @T @T @DT @RT(14)ABForceDigital @RT(0) @T @T @UNKNOWN 0 @F
@F @F
@T
@BEG_Attrib
3 @RT(0) @RT(0) @RT(0)
@END_Attrib
1 0 @F @F @F @F

@Var @RT(24)abForceRobotMoldAreaFree @RT(0) @T @T @DERIVED 0 @T @T @DT @RT(14)ABForceDigital @RT(0) @T @T @UNKNOWN 0 @F
@F @F
@T
@BEG_Attrib
3 @RT(0) @RT(0) @RT(0)
@END_Attrib
1 0 @F @F @F @F

@Var @RT(30)abForceRobotEnableFullMoldOpen @RT(0) @T @T @DERIVED 0 @T @T @DT @RT(14)ABForceDigital @RT(0) @T @T @UNKNOWN 0 @F
@F @F
@T
@BEG_Attrib
3 @RT(0) @RT(0) @RT(0)
@END_Attrib
1 0 @F @F @F @F

@Var @RT(29)abForceRobotEnableMoldClosure @RT(0) @T @T @DERIVED 0 @T @T @DT @RT(14)ABForceDigital @RT(0) @T @T @UNKNOWN 0 @F
@F @F
@T
@BEG_Attrib
3 @RT(0) @RT(0) @RT(0)
@END_Attrib
1 0 @F @F @F @F

@END_Dcl

@END_Export

@BEG_Body

4

@BEG_Export

@BEG_Algo
@ALGORITHM @RT(5)aInit @STRUCTURED_TEXT
@RT(0) @RT(0) @RT(0) @F @F
@END_Algo

@BEG_Dcl
@RT(16)DclTreeContainer
2
@Var @RT(3)bOK @RT(0) @T @F @DT @RT(4)BOOL @RT(0) @T @T @BASIC 0 @F
@F @F
@T
@BEG_Attrib
3 @RT(0) @RT(0) @RT(0)
@END_Attrib
1 3 @F @F @F @F

@Var @RT(12)DeviceString @RT(0) @T @F @DT @RT(11)STRING(255) @RT(0) @T @T @STRING 0 @F @RT(3)255 @F
@F @F
@T
@BEG_Attrib
3 @RT(0) @RT(0) @RT(0)
@END_Attrib
1 0 @F @F @F @F

@END_Dcl

@END_Export

@BEG_Export

@BEG_Algo
@ALGORITHM @RT(8)aCleanup @STRUCTURED_TEXT
@RT(0) @RT(0) @RT(0) @F @F
@END_Algo

@BEG_Dcl
@RT(16)DclTreeContainer
0
@END_Dcl

@END_Export

@BEG_Export

@BEG_Algo
@POSTUPDATE_ALGORITHM @RT(14)pSimulateStart @STRUCTURED_TEXT
@RT(0) @RT(26)sv_bSimulate,sv_bInitStart @RT(9)PU_Task_7 @F @F
@END_Algo

@BEG_Dcl
@RT(16)DclTreeContainer
0
@END_Dcl

@END_Export

@BEG_Export

@BEG_Algo
@PROCESS_ALGORITHM @RT(10)paSimulate @STRUCTURED_TEXT
@RT(0) @RT(0) @RT(7)TaskSim @F @F
@END_Algo

@BEG_Dcl
@RT(16)DclTreeContainer
0
@END_Dcl

@END_Export

@BEG_Body
@TL(21)
mbWantInit := FALSE;
bOK := FALSE;
DeviceString := 'Euromap';

abForceEmergencyStop.aInit(Name := CONCAT(DeviceString, '.di_RobotEmergencyStop'));
abForceRobotOperationMode.aInit(Name := CONCAT(DeviceString, '.di_RobotOperationMode'));

abForceRobotEnableEjectorFwd.aInit(Name := CONCAT(DeviceString, '.di_EnableEjectorFwd'));
abForceRobotEnableEjectorBwd.aInit(Name := CONCAT(DeviceString, '.di_EnableEjectorBwd'));

abForceRobotCore1ToPos1.aInit(Name := CONCAT(DeviceString, '.di_EnableCore1ToPos1'));
abForceRobotCore1ToPos2.aInit(Name := CONCAT(DeviceString, '.di_EnableCore1ToPos2'));
abForceRobotCore2ToPos1.aInit(Name := CONCAT(DeviceString, '.di_EnableCore2ToPos1'));
abForceRobotCore2ToPos2.aInit(Name := CONCAT(DeviceString, '.di_EnableCore2ToPos2'));

abForceRobotMoldAreaFree.aInit(Name := CONCAT(DeviceString, '.di_MoldAreaFree'));
abForceRobotEnableFullMoldOpen.aInit(Name := CONCAT(DeviceString, '.di_EnableFullMoldOpening'));
abForceRobotEnableMoldClosure.aInit(Name := CONCAT(DeviceString, '.di_EnableMoldClosure'));

bOK := TRUE;

@END_Body

@@@BEG_Comment@@@
@TL(0)

@@@END_Comment@@@

@BEG_Body
@TL(17)
mbWantCleanup := FALSE;

abForceEmergencyStop.aUnforce();
abForceRobotOperationMode.aUnforce();

abForceRobotEnableEjectorFwd.aUnforce();
abForceRobotEnableEjectorBwd.aUnforce();

abForceRobotCore1ToPos1.aUnforce();
abForceRobotCore1ToPos2.aUnforce();
abForceRobotCore2ToPos1.aUnforce();
abForceRobotCore2ToPos2.aUnforce();

abForceRobotMoldAreaFree.aUnforce();
abForceRobotEnableFullMoldOpen.aUnforce();
abForceRobotEnableMoldClosure.aUnforce();

@END_Body

@@@BEG_Comment@@@
@TL(0)

@@@END_Comment@@@

@BEG_Body
@TL(8)
IF sv_bSimulate THEN
   mbWantInit := TRUE;
   START_PROCESS_ALGORITHM(paSimulate);
ELSE
   mbWantCleanup := TRUE;
   START_PROCESS_ALGORITHM(paSimulate); //make sure it runs cleanup
END_IF;

@END_Body

@@@BEG_Comment@@@
@TL(0)

@@@END_Comment@@@

@BEG_Body
@TL(33)
IF mbWantInit THEN
   aInit();
   IF NOT aInit.bOK THEN
      STOP_PROCESS_ALGORITHM();
      RETURN;
   END_IF;
END_IF;

//TRUE = emergency stop OK
abForceEmergencyStop.aSetForceValue(bValue := NOT sv_bRobotEmergencyStop);

//FALSE = Operation with injection molding machine
//TRUE  = No operation with injection molding machine
abForceRobotOperationMode.aSetForceValue(bValue := NOT sv_bRobotTurnedOn);

//For now we just simulate that all movements are allowed immediately
abForceRobotEnableEjectorFwd.aSetForceValue(bValue := mbEnableEjectorFwd);
abForceRobotEnableEjectorBwd.aSetForceValue(bValue := mbEnableEjectorBwd);

abForceRobotCore1ToPos1.aSetForceValue(bValue := mbEnableCore1ToPos1);
abForceRobotCore1ToPos2.aSetForceValue(bValue := mbEnableCore1ToPos2);
abForceRobotCore2ToPos1.aSetForceValue(bValue := mbEnableCore2ToPos1);
abForceRobotCore2ToPos2.aSetForceValue(bValue := mbEnableCore2ToPos2);

abForceRobotMoldAreaFree.aSetForceValue(bValue := mbMoldAreaFree);
abForceRobotEnableFullMoldOpen.aSetForceValue(bValue := mbEnableMoldClosure);
abForceRobotEnableMoldClosure.aSetForceValue(bValue := mbEnableFullMoldOpening);

IF mbWantCleanup THEN
   aCleanup();
   STOP_PROCESS_ALGORITHM();
END_IF;

@END_Body

@@@BEG_Comment@@@
@TL(0)

@@@END_Comment@@@
@END_Body

@END_Contents

(* ---- ABForceAnalog.pu ---- *)
IMPORT_OVER_LISTFILE
 KCAT_HandleData
, KCAT_Status
, KSYS_Status
, FBNoiseAI

END_IMPORT

ALGORITHM_BLOCK ABForceAnalog #DUMMY_EDIT_BLOCK

VAR
 Handle : KCAT_HandleData;
 Status : KCAT_Status;
 StatusStatFlag : KSYS_Status;
 mrLastValue : REAL;
 mbLastValueValid : BOOL (* mbLastValue is valid and we do net need to call the forcing routine *);
 mpbStat : REFTO BOOL;
 mRange : REAL;
END_VAR

(*
Initialize the block
and get the reference to the wanted IO endpoint
*)

ALGORITHM aInit

VAR_INPUT
 Name : STRING(255);
 Range : REAL := 10.0;
END_VAR

VAR_OUTPUT
 bOK : BOOL (* init was OK(could get handle for forcing) *);
END_VAR

// VAR_TEMP
 // dummy : DINT;
// END_VAR
#BEGIN_EDIT_BLOCK
(**************************************** WARNING ********************************************
 *** The KEBA Kemro K2 System including software is not intended for safety control tasks! ***
 ***                       For further information see Comment tab!                        ***
 *********************************************************************************************)

bOK := TRUE;
mRange := Range;
Handle := KCAT_GetHandleFromEPName(Name);
IF Handle.Status <> KCAT_Status_OK THEN
   //dummy := Print('simulation: Could not get AI/AO %s for forcing', Name);
   bOK := FALSE;
END_IF;

mpbStat := GET_SYNC_REFTO(SVName := CONCAT(Name, '_stat'), Timeout := t#0S, Status := StatusStatFlag);
IF StatusStatFlag = KSYS_Status_OK THEN
   (* _stat can not be forced, but we can cyclically set it *)
   mpbStat^ := FALSE;
END_IF;

mbLastValueValid := FALSE;

;#END_EDIT_BLOCK END_ALGORITHM

(*
Unforce the endpoint.

*)

ALGORITHM aUnforce

#BEGIN_EDIT_BLOCK
(**************************************** WARNING ********************************************
 *** The KEBA Kemro K2 System including software is not intended for safety control tasks! ***
 ***                       For further information see Comment tab!                        ***
 *********************************************************************************************)

IF Handle.Status = KCAT_Status_OK THEN
   Status := KCAT_UnForce(Handle := Handle.Handle);
END_IF;

mbLastValueValid := FALSE;

;#END_EDIT_BLOCK END_ALGORITHM

(*
Set the force value of the endpoint.
If it was not forced before, forcing is enabled.
If it was forced before the force value is updated.

If a _stat variable exists for the endpoint is is set to FALSE
*)

ALGORITHM aSetForceValue

VAR_INPUT
 rValue : REAL;
END_VAR

VAR_TEMP
 rTmpVal : REAL;
END_VAR

VAR
 fbNoise : FBNoiseAI;
END_VAR
#BEGIN_EDIT_BLOCK
(**************************************** WARNING ********************************************
 *** The KEBA Kemro K2 System including software is not intended for safety control tasks! ***
 ***                       For further information see Comment tab!                        ***
 *********************************************************************************************)

IF Handle.Status = KCAT_Status_OK THEN
   IF StatusStatFlag = KSYS_Status_OK THEN
      (* _stat can not be forced, but we can cyclically set it *)
      mpbStat^ := FALSE;
   END_IF;

   rTmpVal := rValue;
   fbNoise(rTmpVal, mRange);

   IF mbLastValueValid AND mrLastValue = rTmpVal THEN
      (* nothing changed, save some CPU cycles *)
      RETURN;
   END_IF;

   Status := KCAT_SetForceValue(Handle := Handle.Handle,
                                Buffer := rTmpVal);
   mrLastValue := rTmpVal;
   mbLastValueValid := TRUE;
END_IF;

;#END_EDIT_BLOCK END_ALGORITHM

END_ALGORITHM_BLOCK

#END_OF_IEC_PART

@Puma @IecEditor 6 96 @Pou 25
@@@BEG_Comment@@@

@@@END_Comment@@@

@BEG_Contents

@BEG_Func
@RT(17)FuncTreeContainer
0
@END_Func

@BEG_Const
@RT(18)ConstTreeContainer
0
@END_Const

@BEG_Export

@BEG_Kind
@ALGORITHM_BLOCK @RT(13)ABForceAnalog @STRUCTURED_TEXT
@RT(0) @RT(0) @RT(0)
@END_Kind

@BEG_Dcl
@RT(16)DclTreeContainer
7
@Var @RT(6)Handle @RT(0) @T @T @DERIVED 0 @T @T @DT @RT(15)KCAT_HandleData @RT(0) @T @T @UNKNOWN 0 @F
@F @F
@T
@BEG_Attrib
3 @RT(0) @RT(0) @RT(0)
@END_Attrib
1 0 @F @F @F @F

@Var @RT(6)Status @RT(0) @T @T @DERIVED 0 @T @T @DT @RT(11)KCAT_Status @RT(0) @T @T @UNKNOWN 0 @F
@F @F
@T
@BEG_Attrib
3 @RT(0) @RT(0) @RT(0)
@END_Attrib
1 0 @F @F @F @F

@Var @RT(14)StatusStatFlag @RT(0) @T @T @DERIVED 0 @T @T @DT @RT(11)KSYS_Status @RT(0) @T @T @UNKNOWN 0 @F
@F @F
@T
@BEG_Attrib
3 @RT(0) @RT(0) @RT(0)
@END_Attrib
1 0 @F @F @F @F

@Var @RT(11)mrLastValue @RT(0) @T @F @DT @RT(4)REAL @RT(0) @T @T @BASIC 0 @F
@F @F
@T
@BEG_Attrib
3 @RT(0) @RT(0) @RT(0)
@END_Attrib
1 0 @F @F @F @F

@Var @RT(16)mbLastValueValid @RT(0) @T @F @DT @RT(4)BOOL @RT(0) @T @T @BASIC 0 @F
@F @F
@T
@BEG_Attrib
3 @RT(0) @RT(67)mbLastValue is valid and we do net need to call the forcing routine @RT(0)
@END_Attrib
1 0 @F @F @F @F

@Var @RT(7)mpbStat @RT(0) @T @T @REFTO 0 @T @DT @RT(4)BOOL @RT(0) @T @T @BASIC 0 @F
@F @F
@T
@BEG_Attrib
3 @RT(0) @RT(0) @RT(0)
@END_Attrib
1 0 @F @F @F @F

@Var @RT(6)mRange @RT(0) @T @F @DT @RT(4)REAL @RT(0) @T @T @BASIC 0 @F
@F @F
@T
@BEG_Attrib
3 @RT(0) @RT(0) @RT(0)
@END_Attrib
1 0 @F @F @F @F

@END_Dcl

@END_Export

@BEG_Body

3

@BEG_Export

@BEG_Algo
@ALGORITHM @RT(5)aInit @STRUCTURED_TEXT
@RT(0) @RT(0) @RT(0) @F @F
@END_Algo

@BEG_Dcl
@RT(16)DclTreeContainer
4
@Var @RT(4)Name @RT(0) @T @F @DT @RT(11)STRING(255) @RT(0) @T @T @STRING 0 @F @RT(3)255 @F
@F @F
@T
@BEG_Attrib
3 @RT(0) @RT(0) @RT(0)
@END_Attrib
1 1 @F @F @F @F

@Var @RT(5)Range @RT(0) @T @F @DT @RT(4)REAL @RT(0) @T @T @BASIC 0 @F
@F @F
@T
@BEG_Attrib
3 @RT(4)10.0 @RT(0) @RT(0)
@END_Attrib
1 1 @F @F @F @F

@Var @RT(3)bOK @RT(0) @T @F @DT @RT(4)BOOL @RT(0) @T @T @BASIC 0 @F
@F @F
@T
@BEG_Attrib
3 @RT(0) @RT(41)init was OK(could get handle for forcing) @RT(0)
@END_Attrib
1 3 @F @F @F @F

@Var @RT(5)dummy @RT(0) @T @F @DT @RT(4)DINT @RT(0) @T @T @BASIC 0 @F
@F @T
@T
@BEG_Attrib
3 @RT(0) @RT(0) @RT(0)
@END_Attrib
1 4 @F @F @F @F

@END_Dcl

@END_Export

@BEG_Export

@BEG_Algo
@ALGORITHM @RT(8)aUnforce @STRUCTURED_TEXT
@RT(0) @RT(0) @RT(0) @F @F
@END_Algo

@BEG_Dcl
@RT(16)DclTreeContainer
0
@END_Dcl

@END_Export

@BEG_Export

@BEG_Algo
@ALGORITHM @RT(14)aSetForceValue @STRUCTURED_TEXT
@RT(0) @RT(0) @RT(0) @F @F
@END_Algo

@BEG_Dcl
@RT(16)DclTreeContainer
3
@Var @RT(6)rValue @RT(0) @T @F @DT @RT(4)REAL @RT(0) @T @T @BASIC 0 @F
@F @F
@T
@BEG_Attrib
3 @RT(0) @RT(0) @RT(0)
@END_Attrib
1 1 @F @F @F @F

@Var @RT(7)rTmpVal @RT(0) @T @F @DT @RT(4)REAL @RT(0) @T @T @BASIC 0 @F
@F @F
@T
@BEG_Attrib
3 @RT(0) @RT(0) @RT(0)
@END_Attrib
1 4 @F @F @F @F

@Var @RT(7)fbNoise @RT(0) @T @T @DERIVED 0 @F @RT(9)FBNoiseAI @F
@T
@BEG_Attrib
3 @RT(0) @RT(0) @RT(0)
@END_Attrib
1 0 @F @F @F @F

@END_Dcl

@END_Export

@BEG_Body
@TL(21)
(**************************************** WARNING ********************************************
 *** The KEBA Kemro K2 System including software is not intended for safety control tasks! ***
 ***                       For further information see Comment tab!                        ***
 *********************************************************************************************)

bOK := TRUE;
mRange := Range;
Handle := KCAT_GetHandleFromEPName(Name);
IF Handle.Status <> KCAT_Status_OK THEN
   //dummy := Print('simulation: Could not get AI/AO %s for forcing', Name);
   bOK := FALSE;
END_IF;

mpbStat := GET_SYNC_REFTO(SVName := CONCAT(Name, '_stat'), Timeout := t#0S, Status := StatusStatFlag);
IF StatusStatFlag = KSYS_Status_OK THEN
   (* _stat can not be forced, but we can cyclically set it *)
   mpbStat^ := FALSE;
END_IF;

mbLastValueValid := FALSE;

@END_Body

@@@BEG_Comment@@@
@TL(2)
Initialize the block
and get the reference to the wanted IO endpoint
@@@END_Comment@@@

@BEG_Body
@TL(12)
(**************************************** WARNING ********************************************
 *** The KEBA Kemro K2 System including software is not intended for safety control tasks! ***
 ***                       For further information see Comment tab!                        ***
 *********************************************************************************************)

IF Handle.Status = KCAT_Status_OK THEN
   Status := KCAT_UnForce(Handle := Handle.Handle);
END_IF;

mbLastValueValid := FALSE;

@END_Body

@@@BEG_Comment@@@
@TL(2)
Unforce the endpoint.

@@@END_Comment@@@

@BEG_Body
@TL(26)
(**************************************** WARNING ********************************************
 *** The KEBA Kemro K2 System including software is not intended for safety control tasks! ***
 ***                       For further information see Comment tab!                        ***
 *********************************************************************************************)

IF Handle.Status = KCAT_Status_OK THEN
   IF StatusStatFlag = KSYS_Status_OK THEN
      (* _stat can not be forced, but we can cyclically set it *)
      mpbStat^ := FALSE;
   END_IF;

   rTmpVal := rValue;
   fbNoise(rTmpVal, mRange);

   IF mbLastValueValid AND mrLastValue = rTmpVal THEN
      (* nothing changed, save some CPU cycles *)
      RETURN;
   END_IF;

   Status := KCAT_SetForceValue(Handle := Handle.Handle,
                                Buffer := rTmpVal);
   mrLastValue := rTmpVal;
   mbLastValueValid := TRUE;
END_IF;

@END_Body

@@@BEG_Comment@@@
@TL(5)
Set the force value of the endpoint.
If it was not forced before, forcing is enabled.
If it was forced before the force value is updated.

If a _stat variable exists for the endpoint is is set to FALSE
@@@END_Comment@@@
@END_Body

@END_Contents

(* ---- ABForceDigital.pu ---- *)
IMPORT_OVER_LISTFILE
 KCAT_HandleData
, KCAT_Status

END_IMPORT

ALGORITHM_BLOCK ABForceDigital #DUMMY_EDIT_BLOCK

VAR
 Handle : KCAT_HandleData;
 Status : KCAT_Status;
 mbLastValue : BOOL;
 mbLastValueValid : BOOL (* mbLastValue is valid and we do net need to call the forcing routine *);
END_VAR

(*
Initialize the block
and get the reference to the wanted IO endpoint
*)

ALGORITHM aInit

VAR_INPUT
 Name : STRING(255);
END_VAR

VAR_OUTPUT
 bOK : BOOL (* init was OK(could get handle for forcing) *);
END_VAR

// VAR_TEMP
 // dummy : DINT;
// END_VAR
#BEGIN_EDIT_BLOCK
(**************************************** WARNING ********************************************
 *** The KEBA Kemro K2 System including software is not intended for safety control tasks! ***
 ***                       For further information see Comment tab!                        ***
 *********************************************************************************************)

bOK := TRUE;
Handle := KCAT_GetHandleFromEPName(Name);
IF Handle.Status <> KCAT_Status_OK THEN
   //dummy := Print('simulation: Could not get DI/DO %s for forcing', Name);
   bOK := FALSE;
END_IF;
mbLastValueValid := FALSE;

;#END_EDIT_BLOCK END_ALGORITHM

(*
Unforce the endpoint.

*)

ALGORITHM aUnforce

#BEGIN_EDIT_BLOCK
(**************************************** WARNING ********************************************
 *** The KEBA Kemro K2 System including software is not intended for safety control tasks! ***
 ***                       For further information see Comment tab!                        ***
 *********************************************************************************************)

IF Handle.Status = KCAT_Status_OK THEN
   Status := KCAT_UnForce(Handle := Handle.Handle);
END_IF;

mbLastValueValid := FALSE;

;#END_EDIT_BLOCK END_ALGORITHM

(*
Set the force value of the endpoint.
If it was not forced before, forcing is enabled.
If it was forced before the force value is updated.
*)

ALGORITHM aSetForceValue

VAR_INPUT
 bValue : BOOL;
END_VAR

VAR_TEMP
 bTmpVal : BOOL;
END_VAR
#BEGIN_EDIT_BLOCK
(**************************************** WARNING ********************************************
 *** The KEBA Kemro K2 System including software is not intended for safety control tasks! ***
 ***                       For further information see Comment tab!                        ***
 *********************************************************************************************)

IF Handle.Status = KCAT_Status_OK THEN
   IF mbLastValueValid AND mbLastValue = bValue THEN
      (* nothing changed, save some CPU cycles *)
      RETURN;
   END_IF;

   bTmpVal := bValue;
   Status := KCAT_SetForceValue(Handle := Handle.Handle,
                                Buffer := bTmpVal);
   mbLastValue := bTmpVal;
   mbLastValueValid := TRUE;
END_IF;

;#END_EDIT_BLOCK END_ALGORITHM

END_ALGORITHM_BLOCK

#END_OF_IEC_PART

@Puma @IecEditor 6 96 @Pou 25
@@@BEG_Comment@@@

@@@END_Comment@@@

@BEG_Contents

@BEG_Func
@RT(17)FuncTreeContainer
0
@END_Func

@BEG_Const
@RT(18)ConstTreeContainer
0
@END_Const

@BEG_Export

@BEG_Kind
@ALGORITHM_BLOCK @RT(14)ABForceDigital @STRUCTURED_TEXT
@RT(0) @RT(0) @RT(0)
@END_Kind

@BEG_Dcl
@RT(16)DclTreeContainer
4
@Var @RT(6)Handle @RT(0) @T @T @DERIVED 0 @T @T @DT @RT(15)KCAT_HandleData @RT(0) @T @T @UNKNOWN 0 @F
@F @F
@T
@BEG_Attrib
3 @RT(0) @RT(0) @RT(0)
@END_Attrib
1 0 @F @F @F @F

@Var @RT(6)Status @RT(0) @T @T @DERIVED 0 @T @T @DT @RT(11)KCAT_Status @RT(0) @T @T @UNKNOWN 0 @F
@F @F
@T
@BEG_Attrib
3 @RT(0) @RT(0) @RT(0)
@END_Attrib
1 0 @F @F @F @F

@Var @RT(11)mbLastValue @RT(0) @T @F @DT @RT(4)BOOL @RT(0) @T @T @BASIC 0 @F
@F @F
@T
@BEG_Attrib
3 @RT(0) @RT(0) @RT(0)
@END_Attrib
1 0 @F @F @F @F

@Var @RT(16)mbLastValueValid @RT(0) @T @F @DT @RT(4)BOOL @RT(0) @T @T @BASIC 0 @F
@F @F
@T
@BEG_Attrib
3 @RT(0) @RT(67)mbLastValue is valid and we do net need to call the forcing routine @RT(0)
@END_Attrib
1 0 @F @F @F @F

@END_Dcl

@END_Export

@BEG_Body

3

@BEG_Export

@BEG_Algo
@ALGORITHM @RT(5)aInit @STRUCTURED_TEXT
@RT(0) @RT(0) @RT(0) @F @F
@END_Algo

@BEG_Dcl
@RT(16)DclTreeContainer
3
@Var @RT(4)Name @RT(0) @T @F @DT @RT(11)STRING(255) @RT(0) @T @T @STRING 0 @F @RT(3)255 @F
@F @F
@T
@BEG_Attrib
3 @RT(0) @RT(0) @RT(0)
@END_Attrib
1 1 @F @F @F @F

@Var @RT(3)bOK @RT(0) @T @F @DT @RT(4)BOOL @RT(0) @T @T @BASIC 0 @F
@F @F
@T
@BEG_Attrib
3 @RT(0) @RT(41)init was OK(could get handle for forcing) @RT(0)
@END_Attrib
1 3 @F @F @F @F

@Var @RT(5)dummy @RT(0) @T @F @DT @RT(4)DINT @RT(0) @T @T @BASIC 0 @F
@F @T
@T
@BEG_Attrib
3 @RT(0) @RT(0) @RT(0)
@END_Attrib
1 4 @F @F @F @F

@END_Dcl

@END_Export

@BEG_Export

@BEG_Algo
@ALGORITHM @RT(8)aUnforce @STRUCTURED_TEXT
@RT(0) @RT(0) @RT(0) @F @F
@END_Algo

@BEG_Dcl
@RT(16)DclTreeContainer
0
@END_Dcl

@END_Export

@BEG_Export

@BEG_Algo
@ALGORITHM @RT(14)aSetForceValue @STRUCTURED_TEXT
@RT(0) @RT(0) @RT(0) @F @F
@END_Algo

@BEG_Dcl
@RT(16)DclTreeContainer
2
@Var @RT(6)bValue @RT(0) @T @F @DT @RT(4)BOOL @RT(0) @T @T @BASIC 0 @F
@F @F
@T
@BEG_Attrib
3 @RT(0) @RT(0) @RT(0)
@END_Attrib
1 1 @F @F @F @F

@Var @RT(7)bTmpVal @RT(0) @T @F @DT @RT(4)BOOL @RT(0) @T @T @BASIC 0 @F
@F @F
@T
@BEG_Attrib
3 @RT(0) @RT(0) @RT(0)
@END_Attrib
1 4 @F @F @F @F

@END_Dcl

@END_Export

@BEG_Body
@TL(13)
(**************************************** WARNING ********************************************
 *** The KEBA Kemro K2 System including software is not intended for safety control tasks! ***
 ***                       For further information see Comment tab!                        ***
 *********************************************************************************************)

bOK := TRUE;
Handle := KCAT_GetHandleFromEPName(Name);
IF Handle.Status <> KCAT_Status_OK THEN
   //dummy := Print('simulation: Could not get DI/DO %s for forcing', Name);
   bOK := FALSE;
END_IF;
mbLastValueValid := FALSE;

@END_Body

@@@BEG_Comment@@@
@TL(2)
Initialize the block
and get the reference to the wanted IO endpoint
@@@END_Comment@@@

@BEG_Body
@TL(12)
(**************************************** WARNING ********************************************
 *** The KEBA Kemro K2 System including software is not intended for safety control tasks! ***
 ***                       For further information see Comment tab!                        ***
 *********************************************************************************************)

IF Handle.Status = KCAT_Status_OK THEN
   Status := KCAT_UnForce(Handle := Handle.Handle);
END_IF;

mbLastValueValid := FALSE;

@END_Body

@@@BEG_Comment@@@
@TL(2)
Unforce the endpoint.

@@@END_Comment@@@

@BEG_Body
@TL(18)
(**************************************** WARNING ********************************************
 *** The KEBA Kemro K2 System including software is not intended for safety control tasks! ***
 ***                       For further information see Comment tab!                        ***
 *********************************************************************************************)

IF Handle.Status = KCAT_Status_OK THEN
   IF mbLastValueValid AND mbLastValue = bValue THEN
      (* nothing changed, save some CPU cycles *)
      RETURN;
   END_IF;

   bTmpVal := bValue;
   Status := KCAT_SetForceValue(Handle := Handle.Handle,
                                Buffer := bTmpVal);
   mbLastValue := bTmpVal;
   mbLastValueValid := TRUE;
END_IF;

@END_Body

@@@BEG_Comment@@@
@TL(3)
Set the force value of the endpoint.
If it was not forced before, forcing is enabled.
If it was forced before the force value is updated.
@@@END_Comment@@@
@END_Body

@END_Contents
